SPLINE
SPL {X  -141.948, Y  +760.885, Z    +0.000, E1   -42.258, E3 +401984.281}
SPL {X  -160.264, Y  +717.397, Z    +0.000, E1   -24.835, E3 +402025.465}
SPL {X  -164.762, Y  +692.628, Z    +0.000, E1   -12.660, E3 +402028.718}
SPL {X  -165.581, Y  +680.274, Z    +0.000, E1    -5.699, E3 +402024.203}
SPL {X  -165.650, Y  +672.825, Z    +0.000, E1    -0.909, E3 +402022.391}
SPL {X  -165.650, Y  +667.803, Z    +0.000, E1    +2.989, E3 +402021.851}
SPL {X  -165.650, Y  +662.773, Z    +0.000, E1    +7.549, E3 +402021.773}
SPL {X  -165.650, Y  +656.581, Z    +0.000, E1   +13.870, E3 +402019.823}
SPL {X  -165.650, Y  +648.120, Z    +0.000, E1   +22.794, E3 +402019.054}
SPL {X  -165.650, Y  +632.103, Z    +0.000, E1   +42.949, E3 +402006.012}
SPL {X  -165.650, Y  +608.448, Z    +0.000, E1   +47.265, E3 +402032.452}
SPL {X  -165.650, Y  +595.526, Z    +0.000, E1   +48.856, E3 +402046.310}
SPL {X  -165.650, Y  +568.828, Z    +0.000, E1   +48.639, E3 +402088.863}
ENDSPLINE

SPLINE
SPL {X  -165.650, Y  +586.972, Z    +0.000, E1   +40.422, E3 +402099.562}
ENDSPLINE

SPLINE
SPL {X  -165.650, Y  +585.370, Z    +0.000, E1   +38.910, E3 +402112.822}
SPL {X  -165.650, Y  +580.805, Z    +0.000, E1   +38.877, E3 +402124.444}
SPL {X  -165.650, Y  +575.679, Z    +0.000, E1   +38.947, E3 +402137.166}
SPL {X  -165.650, Y  +569.616, Z    +0.000, E1   +38.966, E3 +402152.325}
SPL {X  -165.650, Y  +564.364, Z    +0.000, E1   +38.909, E3 +402165.977}
SPL {X  -165.650, Y  +559.065, Z    +0.000, E1   +38.883, E3 +402179.555}
SPL {X  -165.650, Y  +552.770, Z    +0.000, E1   +38.963, E3 +402195.116}
SPL {X  -165.650, Y  +546.277, Z    +0.000, E1   +38.910, E3 +402211.858}
SPL {X  -165.650, Y  +540.151, Z    +0.000, E1   +38.996, E3 +402226.787}
SPL {X  -165.650, Y  +534.008, Z    +0.000, E1   +38.962, E3 +402242.629}
SPL {X  -165.650, Y  +528.320, Z    +0.000, E1   +38.809, E3 +402257.866}
SPL {X  -165.650, Y  +524.195, Z    +0.000, E1   +38.844, E3 +402268.042}
SPL {X  -165.650, Y  +520.666, Z    +0.000, E1   +39.043, E3 +402275.767}
ENDSPLINE

SPLINE
SPL {X  -165.650, Y  +539.854, Z    +0.000, E1   +28.090, E3 +402288.602}
ENDSPLINE

SPLINE
SPL {X  -165.650, Y  +534.443, Z    +0.000, E1   +28.969, E3 +402302.654}
SPL {X  -165.650, Y  +530.452, Z    +0.000, E1   +29.664, E3 +402312.387}
SPL {X  -165.650, Y  +525.298, Z    +0.000, E1   +30.602, E3 +402324.197}
SPL {X  -165.650, Y  +518.290, Z    +0.000, E1   +31.783, E3 +402340.090}
SPL {X  -165.650, Y  +512.706, Z    +0.000, E1   +32.573, E3 +402352.924}
SPL {X  -165.650, Y  +507.785, Z    +0.000, E1   +33.438, E3 +402362.861}
SPL {X  -165.650, Y  +501.257, Z    +0.000, E1   +34.478, E3 +402376.101}
SPL {X  -165.650, Y  +493.800, Z    +0.000, E1   +35.486, E3 +402391.589}
SPL {X  -165.650, Y  +485.583, Z    +0.000, E1   +36.670, E3 +402407.312}
SPL {X  -165.650, Y  +477.375, Z    +0.000, E1   +37.747, E3 +402422.831}
SPL {X  -165.650, Y  +469.901, Z    +0.000, E1   +38.767, E3 +402435.963}
SPL {X  -165.650, Y  +461.805, Z    +0.000, E1   +39.619, E3 +402451.306}
SPL {X  -165.650, Y  +455.681, Z    +0.000, E1   +39.641, E3 +402466.095}
SPL {X  -165.650, Y  +451.332, Z    +0.000, E1   +39.738, E3 +402476.227}
SPL {X  -165.650, Y  +448.050, Z    +0.000, E1   +39.392, E3 +402486.393}
SPL {X  -165.650, Y  +442.946, Z    +0.000, E1   +39.866, E3 +402496.168}
SPL {X  -165.650, Y  +439.091, Z    +0.000, E1   +39.674, E3 +402506.786}
SPL {X  -165.650, Y  +434.131, Z    +0.000, E1   +39.643, E3 +402519.298}
SPL {X  -165.650, Y  +428.810, Z    +0.000, E1   +39.691, E3 +402532.060}
SPL {X  -165.650, Y  +424.197, Z    +0.000, E1   +39.695, E3 +402543.419}
SPL {X  -165.650, Y  +420.220, Z    +0.000, E1   +39.526, E3 +402554.214}
SPL {X  -165.650, Y  +414.177, Z    +0.000, E1   +39.693, E3 +402568.341}
SPL {X  -165.650, Y  +407.394, Z    +0.000, E1   +39.797, E3 +402584.296}
SPL {X  -165.650, Y  +402.798, Z    +0.000, E1   +39.651, E3 +402596.417}
SPL {X  -165.650, Y  +398.253, Z    +0.000, E1   +39.688, E3 +402607.421}
SPL {X  -165.650, Y  +393.720, Z    +0.000, E1   +39.686, E3 +402618.595}
SPL {X  -165.650, Y  +389.210, Z    +0.000, E1   +39.696, E3 +402629.645}
SPL {X  -165.650, Y  +384.878, Z    +0.000, E1   +39.631, E3 +402640.721}
SPL {X  -165.650, Y  +380.529, Z    +0.000, E1   +39.528, E3 +402652.108}
SPL {X  -165.618, Y  +375.240, Z    +0.000, E1   +39.617, E3 +402664.702}
SPL {X  -165.428, Y  +369.922, Z    +0.000, E1   +39.705, E3 +402677.243}
SPL {X  -165.216, Y  +366.519, Z    +0.000, E1   +39.498, E3 +402686.810}
SPL {X  -164.790, Y  +361.646, Z    +0.000, E1   +39.684, E3 +402697.805}
SPL {X  -164.317, Y  +357.530, Z    +0.000, E1   +39.402, E3 +402709.518}
SPL {X  -163.775, Y  +353.645, Z    +0.000, E1   +39.313, E3 +402719.689}
SPL {X  -162.932, Y  +348.615, Z    +0.000, E1   +39.259, E3 +402732.453}
SPL {X  -162.143, Y  +344.596, Z    +0.000, E1   +39.019, E3 +402743.670}
SPL {X  -161.093, Y  +339.912, Z    +0.000, E1   +38.966, E3 +402755.620}
SPL {X  -159.926, Y  +335.332, Z    +0.000, E1   +38.809, E3 +402767.674}
SPL {X  -154.584, Y  +318.971, Z    +0.000, E1   +44.936, E3 +402770.305}
SPL {X  -151.650, Y  +311.851, Z    +0.000, E1   +46.071, E3 +402777.840}
SPL {X  -148.632, Y  +305.368, Z    +0.000, E1   +40.700, E3 +402834.007}
SPL {X  -145.004, Y  +298.414, Z    +0.000, E1   +40.971, E3 +402858.743}
ENDSPLINE

SPLINE
SPL {X  -149.687, Y  +307.551, Z    +0.000, E1   +36.303, E3 +402894.175}
SPL {X  -158.807, Y  +331.381, Z    +0.000, E1   +26.928, E3 +402917.827}
SPL {X  -164.505, Y  +359.058, Z    +0.000, E1   +13.887, E3 +402906.589}
SPL {X  -165.494, Y  +371.321, Z    +0.000, E1    +7.176, E3 +402905.150}
SPL {X  -165.650, Y  +379.419, Z    +0.000, E1    +2.065, E3 +402902.831}
SPL {X  -165.650, Y  +383.176, Z    +0.000, E1    -0.610, E3 +402903.826}
SPL {X  -165.650, Y  +387.435, Z    +0.000, E1    -4.104, E3 +402902.186}
SPL {X  -165.650, Y  +393.422, Z    +0.000, E1    -9.605, E3 +402902.744}
SPL {X  -165.650, Y  +400.450, Z    +0.000, E1   -18.287, E3 +402894.558}
SPL {X  -165.650, Y  +409.248, Z    +0.000, E1   -26.478, E3 +402898.181}
SPL {X  -165.650, Y  +418.660, Z    +0.000, E1   -36.186, E3 +402895.657}
SPL {X  -165.650, Y  +444.260, Z    +0.000, E1   -47.328, E3 +402911.405}
SPL {X  -165.650, Y  +458.981, Z    +0.000, E1   -49.189, E3 +402926.948}
SPL {X  -165.650, Y  +493.049, Z    +0.000, E1   -51.657, E3 +402965.981}
ENDSPLINE

SPLINE
SPL {X  -165.650, Y  +468.984, Z    +0.000, E1   -41.461, E3 +402978.841}
SPL {X  -165.650, Y  +467.052, Z    +0.000, E1   -38.928, E3 +402989.456}
ENDSPLINE

SPLINE
SPL {X  -165.650, Y  +471.956, Z    +0.000, E1   -39.047, E3 +403001.107}
SPL {X  -165.650, Y  +476.270, Z    +0.000, E1   -39.142, E3 +403011.364}
SPL {X  -165.650, Y  +480.876, Z    +0.000, E1   -39.050, E3 +403023.646}
SPL {X  -165.650, Y  +487.054, Z    +0.000, E1   -39.118, E3 +403038.785}
SPL {X  -165.650, Y  +493.422, Z    +0.000, E1   -39.176, E3 +403054.507}
SPL {X  -165.650, Y  +499.941, Z    +0.000, E1   -39.068, E3 +403071.558}
SPL {X  -165.650, Y  +505.989, Z    +0.000, E1   -39.067, E3 +403086.738}
SPL {X  -165.650, Y  +512.188, Z    +0.000, E1   -39.077, E3 +403102.380}
SPL {X  -165.650, Y  +516.634, Z    +0.000, E1   -39.035, E3 +403113.626}
SPL {X  -165.650, Y  +521.541, Z    +0.000, E1   -39.052, E3 +403126.173}
SPL {X  -165.650, Y  +527.474, Z    +0.000, E1   -39.169, E3 +403140.191}
SPL {X  -165.650, Y  +532.836, Z    +0.000, E1   -39.150, E3 +403153.973}
SPL {X  -165.650, Y  +537.667, Z    +0.000, E1   -38.986, E3 +403166.918}
SPL {X  -165.650, Y  +541.183, Z    +0.000, E1   -39.101, E3 +403175.105}
SPL {X  -165.650, Y  +546.018, Z    +0.000, E1   -39.065, E3 +403187.616}
SPL {X  -165.650, Y  +551.666, Z    +0.000, E1   -39.102, E3 +403201.565}
SPL {X  -165.650, Y  +557.612, Z    +0.000, E1   -39.166, E3 +403216.211}
SPL {X  -165.650, Y  +562.850, Z    +0.000, E1   -38.959, E3 +403230.570}
SPL {X  -165.650, Y  +568.257, Z    +0.000, E1   -39.077, E3 +403243.525}
SPL {X  -165.650, Y  +573.200, Z    +0.000, E1   -39.061, E3 +403256.060}
SPL {X  -165.650, Y  +578.240, Z    +0.000, E1   -39.117, E3 +403268.401}
SPL {X  -165.650, Y  +582.804, Z    +0.000, E1   -39.080, E3 +403280.108}
SPL {X  -165.650, Y  +587.640, Z    +0.000, E1   -39.069, E3 +403292.365}
SPL {X  -165.650, Y  +593.610, Z    +0.000, E1   -39.204, E3 +403306.639}
SPL {X  -165.650, Y  +599.021, Z    +0.000, E1   -38.950, E3 +403321.788}
SPL {X  -165.650, Y  +604.635, Z    +0.000, E1   -39.163, E3 +403334.565}
SPL {X  -165.650, Y  +608.365, Z    +0.000, E1   -39.063, E3 +403344.555}
SPL {X  -165.650, Y  +612.142, Z    +0.000, E1   -39.023, E3 +403354.285}
SPL {X  -165.650, Y  +616.635, Z    +0.000, E1   -39.260, E3 +403364.172}
SPL {X  -165.650, Y  +620.299, Z    +0.000, E1   -38.904, E3 +403375.559}
SPL {X  -165.650, Y  +625.662, Z    +0.000, E1   -39.189, E3 +403387.370}
SPL {X  -165.650, Y  +629.982, Z    +0.000, E1   -39.063, E3 +403398.971}
SPL {X  -165.650, Y  +634.317, Z    +0.000, E1   -39.239, E3 +403408.762}
SPL {X  -165.650, Y  +639.215, Z    +0.000, E1   -39.074, E3 +403422.287}
SPL {X  -165.650, Y  +643.707, Z    +0.000, E1   -38.911, E3 +403434.387}
SPL {X  -165.650, Y  +648.294, Z    +0.000, E1   -39.142, E3 +403444.643}
SPL {X  -165.650, Y  +652.477, Z    +0.000, E1   -39.068, E3 +403455.545}
SPL {X  -165.650, Y  +656.920, Z    +0.000, E1   -39.120, E3 +403466.500}
SPL {X  -165.650, Y  +662.945, Z    +0.000, E1   -39.141, E3 +403481.605}
SPL {X  -165.650, Y  +668.296, Z    +0.000, E1   -39.077, E3 +403495.330}
SPL {X  -165.650, Y  +674.193, Z    +0.000, E1   -39.034, E3 +403510.672}
SPL {X  -165.521, Y  +682.029, Z    +0.000, E1   -39.160, E3 +403529.640}
SPL {X  -165.241, Y  +687.126, Z    +0.000, E1   -39.221, E3 +403541.802}
SPL {X  -164.948, Y  +690.736, Z    +0.000, E1   -38.951, E3 +403552.654}
SPL {X  -164.363, Y  +696.109, Z    +0.000, E1   -38.853, E3 +403566.745}
SPL {X  -163.795, Y  +700.218, Z    +0.000, E1   -38.698, E3 +403577.952}
SPL {X  -162.937, Y  +705.358, Z    +0.000, E1   -38.703, E3 +403591.020}
SPL {X  -161.983, Y  +710.160, Z    +0.000, E1   -38.439, E3 +403604.514}
SPL {X  -161.163, Y  +713.794, Z    +0.000, E1   -38.390, E3 +403613.884}
SPL {X  -160.616, Y  +716.027, Z    +0.000, E1   -37.944, E3 +403622.086}
SPL {X  -158.364, Y  +724.087, Z    +0.000, E1   -39.961, E3 +403630.382}
SPL {X  -138.706, Y  +766.057, Z    +0.000, E1   -46.957, E3 +403681.373}
ENDSPLINE

SPLINE
SPL {X  -141.948, Y  +760.885, Z    +0.000, E1   -42.258, E3 +403721.123}
SPL {X  -152.484, Y  +740.219, Z    +0.000, E1   -33.928, E3 +403758.276}
SPL {X  -161.203, Y  +713.624, Z    +0.000, E1   -23.097, E3 +403762.692}
SPL {X  -164.762, Y  +692.628, Z    +0.000, E1   -12.660, E3 +403765.560}
SPL {X  -165.581, Y  +680.274, Z    +0.000, E1    -5.699, E3 +403761.045}
SPL {X  -165.650, Y  +672.825, Z    +0.000, E1    -0.909, E3 +403759.234}
SPL {X  -165.650, Y  +667.803, Z    +0.000, E1    +2.989, E3 +403758.694}
SPL {X  -165.650, Y  +662.773, Z    +0.000, E1    +7.549, E3 +403758.615}
SPL {X  -165.650, Y  +656.581, Z    +0.000, E1   +13.870, E3 +403756.665}
SPL {X  -165.650, Y  +648.120, Z    +0.000, E1   +22.794, E3 +403755.896}
SPL {X  -165.650, Y  +632.103, Z    +0.000, E1   +42.949, E3 +403742.854}
SPL {X  -165.650, Y  +608.448, Z    +0.000, E1   +47.265, E3 +403769.294}
SPL {X  -165.650, Y  +595.526, Z    +0.000, E1   +48.856, E3 +403783.152}
SPL {X  -165.650, Y  +568.828, Z    +0.000, E1   +48.639, E3 +403825.705}
ENDSPLINE

SPLINE
SPL {X  -165.650, Y  +586.972, Z    +0.000, E1   +40.422, E3 +403836.404}
ENDSPLINE

SPLINE
SPL {X  -165.650, Y  +585.370, Z    +0.000, E1   +38.910, E3 +403849.664}
SPL {X  -165.650, Y  +580.805, Z    +0.000, E1   +38.877, E3 +403861.286}
SPL {X  -165.650, Y  +575.679, Z    +0.000, E1   +38.947, E3 +403874.009}
SPL {X  -165.650, Y  +569.616, Z    +0.000, E1   +38.966, E3 +403889.167}
SPL {X  -165.650, Y  +564.364, Z    +0.000, E1   +38.909, E3 +403902.820}
SPL {X  -165.650, Y  +559.065, Z    +0.000, E1   +38.883, E3 +403916.397}
SPL {X  -165.650, Y  +554.358, Z    +0.000, E1   +38.887, E3 +403928.239}
SPL {X  -165.650, Y  +549.409, Z    +0.000, E1   +38.884, E3 +403940.920}
SPL {X  -165.650, Y  +544.480, Z    +0.000, E1   +38.998, E3 +403952.584}
SPL {X  -165.650, Y  +540.151, Z    +0.000, E1   +38.996, E3 +403963.630}
SPL {X  -165.650, Y  +534.008, Z    +0.000, E1   +38.962, E3 +403979.472}
SPL {X  -165.650, Y  +528.320, Z    +0.000, E1   +38.809, E3 +403994.708}
SPL {X  -165.650, Y  +524.195, Z    +0.000, E1   +38.844, E3 +404004.884}
SPL {X  -165.650, Y  +520.666, Z    +0.000, E1   +39.043, E3 +404012.610}
ENDSPLINE

SPLINE
SPL {X  -165.650, Y  +541.168, Z    +0.000, E1   +27.957, E3 +404021.167}
ENDSPLINE

SPLINE
SPL {X  -165.650, Y  +536.052, Z    +0.000, E1   +28.653, E3 +404035.802}
SPL {X  -165.650, Y  +530.452, Z    +0.000, E1   +29.664, E3 +404049.229}
SPL {X  -165.650, Y  +523.712, Z    +0.000, E1   +30.911, E3 +404064.511}
SPL {X  -165.650, Y  +516.975, Z    +0.000, E1   +31.942, E3 +404080.105}
SPL {X  -165.650, Y  +512.706, Z    +0.000, E1   +32.573, E3 +404089.766}
SPL {X  -165.650, Y  +507.785, Z    +0.000, E1   +33.438, E3 +404099.703}
SPL {X  -165.650, Y  +501.257, Z    +0.000, E1   +34.478, E3 +404112.943}
SPL {X  -165.650, Y  +495.236, Z    +0.000, E1   +35.288, E3 +404125.449}
SPL {X  -165.650, Y  +488.684, Z    +0.000, E1   +36.217, E3 +404138.345}
SPL {X  -165.650, Y  +481.130, Z    +0.000, E1   +37.251, E3 +404152.654}
SPL {X  -165.650, Y  +475.455, Z    +0.000, E1   +37.964, E3 +404163.311}
SPL {X  -165.650, Y  +469.901, Z    +0.000, E1   +38.767, E3 +404172.805}
SPL {X  -165.650, Y  +465.276, Z    +0.000, E1   +39.067, E3 +404182.682}
SPL {X  -165.650, Y  +459.623, Z    +0.000, E1   +39.919, E3 +404191.617}
SPL {X  -165.650, Y  +455.681, Z    +0.000, E1   +39.641, E3 +404202.937}
SPL {X  -165.650, Y  +451.332, Z    +0.000, E1   +39.738, E3 +404213.069}
SPL {X  -165.650, Y  +448.050, Z    +0.000, E1   +39.392, E3 +404223.235}
SPL {X  -165.650, Y  +442.946, Z    +0.000, E1   +39.866, E3 +404233.010}
SPL {X  -165.650, Y  +439.091, Z    +0.000, E1   +39.674, E3 +404243.628}
SPL {X  -165.650, Y  +435.404, Z    +0.000, E1   +39.549, E3 +404253.465}
SPL {X  -165.650, Y  +429.757, Z    +0.000, E1   +39.737, E3 +404266.414}
SPL {X  -165.650, Y  +424.197, Z    +0.000, E1   +39.695, E3 +404280.261}
SPL {X  -165.650, Y  +420.220, Z    +0.000, E1   +39.526, E3 +404291.056}
SPL {X  -165.650, Y  +415.675, Z    +0.000, E1   +39.706, E3 +404301.218}
SPL {X  -165.650, Y  +410.648, Z    +0.000, E1   +39.653, E3 +404314.019}
SPL {X  -165.650, Y  +403.851, Z    +0.000, E1   +39.774, E3 +404330.104}
SPL {X  -165.650, Y  +398.253, Z    +0.000, E1   +39.688, E3 +404344.263}
SPL {X  -165.650, Y  +393.720, Z    +0.000, E1   +39.686, E3 +404355.437}
SPL {X  -165.650, Y  +389.210, Z    +0.000, E1   +39.696, E3 +404366.487}
SPL {X  -165.650, Y  +384.878, Z    +0.000, E1   +39.631, E3 +404377.564}
SPL {X  -165.650, Y  +380.529, Z    +0.000, E1   +39.528, E3 +404388.950}
SPL {X  -165.618, Y  +375.240, Z    +0.000, E1   +39.617, E3 +404401.544}
SPL {X  -165.428, Y  +369.922, Z    +0.000, E1   +39.705, E3 +404414.086}
SPL {X  -165.055, Y  +364.469, Z    +0.000, E1   +39.623, E3 +404428.127}
SPL {X  -164.424, Y  +358.387, Z    +0.000, E1   +39.525, E3 +404443.651}
SPL {X  -163.775, Y  +353.645, Z    +0.000, E1   +39.313, E3 +404456.531}
SPL {X  -162.932, Y  +348.615, Z    +0.000, E1   +39.259, E3 +404469.295}
SPL {X  -161.858, Y  +343.258, Z    +0.000, E1   +39.040, E3 +404483.834}
SPL {X  -160.812, Y  +338.758, Z    +0.000, E1   +38.898, E3 +404495.559}
SPL {X  -159.926, Y  +335.332, Z    +0.000, E1   +38.809, E3 +404504.516}
SPL {X  -153.020, Y  +315.059, Z    +0.000, E1   +45.580, E3 +404511.248}
SPL {X  -148.632, Y  +305.368, Z    +0.000, E1   +40.700, E3 +404570.849}
SPL {X  -145.004, Y  +298.414, Z    +0.000, E1   +40.971, E3 +404595.585}
ENDSPLINE

SPLINE
SPL {X  -149.687, Y  +307.551, Z    +0.000, E1   +36.303, E3 +404631.017}
SPL {X  -158.807, Y  +331.381, Z    +0.000, E1   +26.928, E3 +404654.670}
SPL {X  -164.505, Y  +359.058, Z    +0.000, E1   +13.887, E3 +404643.431}
SPL {X  -165.334, Y  +368.271, Z    +0.000, E1    +8.886, E3 +404641.270}
SPL {X  -165.596, Y  +374.277, Z    +0.000, E1    +5.306, E3 +404642.652}
SPL {X  -165.650, Y  +379.419, Z    +0.000, E1    +2.065, E3 +404639.673}
SPL {X  -165.650, Y  +383.176, Z    +0.000, E1    -0.610, E3 +404640.668}
SPL {X  -165.650, Y  +387.435, Z    +0.000, E1    -4.104, E3 +404639.029}
SPL {X  -165.650, Y  +393.422, Z    +0.000, E1    -9.605, E3 +404639.586}
SPL {X  -165.650, Y  +400.450, Z    +0.000, E1   -18.287, E3 +404631.400}
SPL {X  -165.650, Y  +409.248, Z    +0.000, E1   -26.478, E3 +404635.023}
SPL {X  -165.650, Y  +418.660, Z    +0.000, E1   -36.186, E3 +404632.499}
SPL {X  -165.650, Y  +444.260, Z    +0.000, E1   -47.328, E3 +404648.247}
SPL {X  -165.650, Y  +458.981, Z    +0.000, E1   -49.189, E3 +404663.791}
SPL {X  -165.650, Y  +493.049, Z    +0.000, E1   -51.657, E3 +404702.823}
ENDSPLINE

SPLINE
SPL {X  -165.650, Y  +468.984, Z    +0.000, E1   -41.461, E3 +404715.684}
SPL {X  -165.650, Y  +467.052, Z    +0.000, E1   -38.928, E3 +404726.298}
ENDSPLINE

SPLINE
SPL {X  -165.650, Y  +471.956, Z    +0.000, E1   -39.047, E3 +404737.949}
SPL {X  -165.650, Y  +476.270, Z    +0.000, E1   -39.142, E3 +404748.206}
SPL {X  -165.650, Y  +479.585, Z    +0.000, E1   -39.047, E3 +404757.117}
SPL {X  -165.650, Y  +484.115, Z    +0.000, E1   -39.050, E3 +404768.595}
SPL {X  -165.650, Y  +490.374, Z    +0.000, E1   -39.169, E3 +404783.715}
SPL {X  -165.650, Y  +495.141, Z    +0.000, E1   -39.109, E3 +404795.871}
SPL {X  -165.650, Y  +497.824, Z    +0.000, E1   -38.944, E3 +404803.630}
SPL {X  -165.650, Y  +502.351, Z    +0.000, E1   -39.056, E3 +404814.513}
SPL {X  -165.650, Y  +508.180, Z    +0.000, E1   -39.157, E3 +404828.579}
SPL {X  -165.650, Y  +513.074, Z    +0.000, E1   -38.997, E3 +404841.796}
SPL {X  -165.650, Y  +518.439, Z    +0.000, E1   -39.071, E3 +404854.947}
SPL {X  -165.650, Y  +523.032, Z    +0.000, E1   -38.966, E3 +404867.083}
SPL {X  -165.650, Y  +528.401, Z    +0.000, E1   -39.135, E3 +404879.683}
SPL {X  -165.650, Y  +533.857, Z    +0.000, E1   -39.163, E3 +404893.189}
SPL {X  -165.650, Y  +539.651, Z    +0.000, E1   -39.087, E3 +404908.333}
SPL {X  -165.650, Y  +544.603, Z    +0.000, E1   -39.103, E3 +404920.509}
SPL {X  -165.650, Y  +547.280, Z    +0.000, E1   -38.965, E3 +404928.089}
SPL {X  -165.650, Y  +551.666, Z    +0.000, E1   -39.102, E3 +404938.407}
SPL {X  -165.650, Y  +555.880, Z    +0.000, E1   -39.094, E3 +404948.978}
SPL {X  -165.650, Y  +559.255, Z    +0.000, E1   -39.167, E3 +404957.014}
SPL {X  -165.650, Y  +562.850, Z    +0.000, E1   -38.959, E3 +404967.412}
SPL {X  -165.650, Y  +568.257, Z    +0.000, E1   -39.077, E3 +404980.367}
SPL {X  -165.650, Y  +573.200, Z    +0.000, E1   -39.061, E3 +404992.902}
SPL {X  -165.650, Y  +578.240, Z    +0.000, E1   -39.117, E3 +405005.243}
SPL {X  -165.650, Y  +582.804, Z    +0.000, E1   -39.080, E3 +405016.950}
SPL {X  -165.650, Y  +587.640, Z    +0.000, E1   -39.069, E3 +405029.207}
SPL {X  -165.650, Y  +592.685, Z    +0.000, E1   -39.263, E3 +405040.671}
SPL {X  -165.650, Y  +596.539, Z    +0.000, E1   -39.049, E3 +405051.661}
SPL {X  -165.650, Y  +599.973, Z    +0.000, E1   -38.814, E3 +405061.714}
SPL {X  -165.650, Y  +604.635, Z    +0.000, E1   -39.163, E3 +405071.407}
SPL {X  -165.650, Y  +608.365, Z    +0.000, E1   -39.063, E3 +405081.397}
SPL {X  -165.650, Y  +612.142, Z    +0.000, E1   -39.023, E3 +405091.127}
SPL {X  -165.650, Y  +616.635, Z    +0.000, E1   -39.260, E3 +405101.014}
SPL {X  -165.650, Y  +620.299, Z    +0.000, E1   -38.904, E3 +405112.401}
SPL {X  -165.650, Y  +625.662, Z    +0.000, E1   -39.189, E3 +405124.212}
SPL {X  -165.650, Y  +629.982, Z    +0.000, E1   -39.063, E3 +405135.813}
SPL {X  -165.650, Y  +635.019, Z    +0.000, E1   -39.106, E3 +405148.295}
SPL {X  -165.650, Y  +640.403, Z    +0.000, E1   -39.127, E3 +405161.691}
SPL {X  -165.650, Y  +643.707, Z    +0.000, E1   -38.911, E3 +405171.229}
SPL {X  -165.650, Y  +648.294, Z    +0.000, E1   -39.142, E3 +405181.485}
SPL {X  -165.650, Y  +652.477, Z    +0.000, E1   -39.068, E3 +405192.387}
SPL {X  -165.650, Y  +656.920, Z    +0.000, E1   -39.120, E3 +405203.342}
SPL {X  -165.650, Y  +662.945, Z    +0.000, E1   -39.141, E3 +405218.448}
SPL {X  -165.650, Y  +668.296, Z    +0.000, E1   -39.077, E3 +405232.172}
SPL {X  -165.650, Y  +674.193, Z    +0.000, E1   -39.034, E3 +405247.514}
SPL {X  -165.521, Y  +682.029, Z    +0.000, E1   -39.160, E3 +405266.483}
SPL {X  -165.241, Y  +687.126, Z    +0.000, E1   -39.221, E3 +405278.644}
SPL {X  -165.072, Y  +689.330, Z    +0.000, E1   -38.812, E3 +405286.692}
SPL {X  -164.582, Y  +694.282, Z    +0.000, E1   -38.975, E3 +405298.301}
SPL {X  -163.926, Y  +699.336, Z    +0.000, E1   -38.767, E3 +405312.279}
SPL {X  -163.214, Y  +703.806, Z    +0.000, E1   -38.755, E3 +405323.464}
SPL {X  -162.700, Y  +706.623, Z    +0.000, E1   -38.580, E3 +405331.576}
SPL {X  -161.983, Y  +710.160, Z    +0.000, E1   -38.439, E3 +405341.356}
SPL {X  -161.163, Y  +713.794, Z    +0.000, E1   -38.390, E3 +405350.726}
SPL {X  -160.158, Y  +717.801, Z    +0.000, E1   -38.225, E3 +405361.856}
SPL {X  -155.870, Y  +731.575, Z    +0.000, E1   -42.661, E3 +405369.319}
SPL {X  -137.799, Y  +767.431, Z    +0.000, E1   -46.550, E3 +405425.829}
ENDSPLINE

SPLINE
SPL {X  -141.948, Y  +760.885, Z    +0.000, E1   -42.258, E3 +405457.965}
SPL {X  -152.484, Y  +740.219, Z    +0.000, E1   -33.928, E3 +405495.119}
SPL {X  -161.203, Y  +713.624, Z    +0.000, E1   -23.097, E3 +405499.534}
SPL {X  -164.762, Y  +692.628, Z    +0.000, E1   -12.660, E3 +405502.402}
SPL {X  -165.481, Y  +682.990, Z    +0.000, E1    -7.255, E3 +405499.247}
SPL {X  -165.649, Y  +676.021, Z    +0.000, E1    -3.061, E3 +405496.614}
SPL {X  -165.650, Y  +670.589, Z    +0.000, E1    +0.778, E3 +405495.851}
SPL {X  -165.650, Y  +666.842, Z    +0.000, E1    +3.871, E3 +405495.312}
SPL {X  -165.650, Y  +662.773, Z    +0.000, E1    +7.549, E3 +405495.457}
SPL {X  -165.650, Y  +656.581, Z    +0.000, E1   +13.870, E3 +405493.507}
SPL {X  -165.650, Y  +648.120, Z    +0.000, E1   +22.794, E3 +405492.738}
SPL {X  -165.650, Y  +632.103, Z    +0.000, E1   +42.949, E3 +405479.696}
SPL {X  -165.650, Y  +608.448, Z    +0.000, E1   +47.265, E3 +405506.136}
SPL {X  -165.650, Y  +595.526, Z    +0.000, E1   +48.856, E3 +405519.994}
SPL {X  -165.650, Y  +568.828, Z    +0.000, E1   +48.639, E3 +405562.547}
ENDSPLINE

SPLINE
SPL {X  -165.650, Y  +586.972, Z    +0.000, E1   +40.422, E3 +405573.246}
ENDSPLINE

SPLINE
SPL {X  -165.650, Y  +585.370, Z    +0.000, E1   +38.910, E3 +405586.506}
SPL {X  -165.650, Y  +580.805, Z    +0.000, E1   +38.877, E3 +405598.128}
SPL {X  -165.650, Y  +575.679, Z    +0.000, E1   +38.947, E3 +405610.851}
SPL {X  -165.650, Y  +569.616, Z    +0.000, E1   +38.966, E3 +405626.009}
SPL {X  -165.650, Y  +564.364, Z    +0.000, E1   +38.909, E3 +405639.662}
SPL {X  -165.650, Y  +559.065, Z    +0.000, E1   +38.883, E3 +405653.240}
SPL {X  -165.650, Y  +552.770, Z    +0.000, E1   +38.963, E3 +405668.800}
SPL {X  -165.650, Y  +546.277, Z    +0.000, E1   +38.910, E3 +405685.542}
SPL {X  -165.650, Y  +541.194, Z    +0.000, E1   +39.037, E3 +405697.475}
SPL {X  -165.650, Y  +537.647, Z    +0.000, E1   +38.838, E3 +405707.720}
SPL {X  -165.650, Y  +532.636, Z    +0.000, E1   +39.009, E3 +405719.366}
SPL {X  -165.650, Y  +528.320, Z    +0.000, E1   +38.809, E3 +405731.550}
SPL {X  -165.650, Y  +522.377, Z    +0.000, E1   +38.974, E3 +405745.670}
ENDSPLINE

SPLINE
SPL {X  -165.650, Y  +541.168, Z    +0.000, E1   +27.957, E3 +405758.010}
ENDSPLINE

SPLINE
SPL {X  -165.650, Y  +536.052, Z    +0.000, E1   +28.653, E3 +405772.644}
SPL {X  -165.650, Y  +530.452, Z    +0.000, E1   +29.664, E3 +405786.071}
SPL {X  -165.650, Y  +523.712, Z    +0.000, E1   +30.911, E3 +405801.353}
SPL {X  -165.650, Y  +516.975, Z    +0.000, E1   +31.942, E3 +405816.947}
SPL {X  -165.650, Y  +512.706, Z    +0.000, E1   +32.573, E3 +405826.608}
SPL {X  -165.650, Y  +507.785, Z    +0.000, E1   +33.438, E3 +405836.546}
SPL {X  -165.650, Y  +502.877, Z    +0.000, E1   +34.230, E3 +405846.434}
SPL {X  -165.650, Y  +496.704, Z    +0.000, E1   +35.113, E3 +405859.227}
SPL {X  -165.650, Y  +488.684, Z    +0.000, E1   +36.217, E3 +405875.188}
SPL {X  -165.650, Y  +481.130, Z    +0.000, E1   +37.251, E3 +405889.497}
SPL {X  -165.650, Y  +475.455, Z    +0.000, E1   +37.964, E3 +405900.153}
SPL {X  -165.650, Y  +469.901, Z    +0.000, E1   +38.767, E3 +405909.647}
SPL {X  -165.650, Y  +461.805, Z    +0.000, E1   +39.619, E3 +405924.990}
SPL {X  -165.650, Y  +455.681, Z    +0.000, E1   +39.641, E3 +405939.779}
SPL {X  -165.650, Y  +451.332, Z    +0.000, E1   +39.738, E3 +405949.912}
SPL {X  -165.650, Y  +448.050, Z    +0.000, E1   +39.392, E3 +405960.077}
SPL {X  -165.650, Y  +442.946, Z    +0.000, E1   +39.866, E3 +405969.852}
SPL {X  -165.650, Y  +439.091, Z    +0.000, E1   +39.674, E3 +405980.470}
SPL {X  -165.650, Y  +434.131, Z    +0.000, E1   +39.643, E3 +405992.983}
SPL {X  -165.650, Y  +428.810, Z    +0.000, E1   +39.691, E3 +406005.745}
SPL {X  -165.650, Y  +424.197, Z    +0.000, E1   +39.695, E3 +406017.103}
SPL {X  -165.650, Y  +420.220, Z    +0.000, E1   +39.526, E3 +406027.898}
SPL {X  -165.650, Y  +414.177, Z    +0.000, E1   +39.693, E3 +406042.025}
SPL {X  -165.650, Y  +407.394, Z    +0.000, E1   +39.797, E3 +406057.980}
SPL {X  -165.650, Y  +402.798, Z    +0.000, E1   +39.651, E3 +406070.102}
SPL {X  -165.650, Y  +398.253, Z    +0.000, E1   +39.688, E3 +406081.105}
SPL {X  -165.650, Y  +393.720, Z    +0.000, E1   +39.686, E3 +406092.280}
SPL {X  -165.650, Y  +389.210, Z    +0.000, E1   +39.696, E3 +406103.329}
SPL {X  -165.650, Y  +384.878, Z    +0.000, E1   +39.631, E3 +406114.406}
SPL {X  -165.650, Y  +378.931, Z    +0.000, E1   +39.598, E3 +406129.502}
SPL {X  -165.490, Y  +371.216, Z    +0.000, E1   +39.708, E3 +406147.874}
SPL {X  -165.055, Y  +364.469, Z    +0.000, E1   +39.623, E3 +406164.969}
SPL {X  -164.424, Y  +358.387, Z    +0.000, E1   +39.525, E3 +406180.493}
SPL {X  -163.775, Y  +353.645, Z    +0.000, E1   +39.313, E3 +406193.373}
SPL {X  -162.932, Y  +348.615, Z    +0.000, E1   +39.259, E3 +406206.137}
SPL {X  -162.143, Y  +344.596, Z    +0.000, E1   +39.019, E3 +406217.354}
SPL {X  -161.093, Y  +339.912, Z    +0.000, E1   +38.966, E3 +406229.305}
SPL {X  -159.926, Y  +335.332, Z    +0.000, E1   +38.809, E3 +406241.358}
SPL {X  -153.020, Y  +315.059, Z    +0.000, E1   +45.580, E3 +406248.090}
SPL {X  -148.632, Y  +305.368, Z    +0.000, E1   +40.700, E3 +406307.692}
SPL {X  -145.004, Y  +298.414, Z    +0.000, E1   +40.971, E3 +406332.427}
ENDSPLINE

SPLINE
SPL {X  -149.687, Y  +307.551, Z    +0.000, E1   +36.303, E3 +406367.859}
SPL {X  -158.807, Y  +331.381, Z    +0.000, E1   +26.928, E3 +406391.512}
SPL {X  -164.505, Y  +359.058, Z    +0.000, E1   +13.887, E3 +406380.274}
SPL {X  -165.494, Y  +371.321, Z    +0.000, E1    +7.176, E3 +406378.834}
SPL {X  -165.650, Y  +379.419, Z    +0.000, E1    +2.065, E3 +406376.516}
SPL {X  -165.650, Y  +383.176, Z    +0.000, E1    -0.610, E3 +406377.511}
SPL {X  -165.650, Y  +388.696, Z    +0.000, E1    -5.134, E3 +406375.787}
SPL {X  -165.650, Y  +394.663, Z    +0.000, E1   -10.843, E3 +406376.943}
SPL {X  -165.650, Y  +400.450, Z    +0.000, E1   -18.287, E3 +406368.242}
SPL {X  -165.650, Y  +409.248, Z    +0.000, E1   -26.478, E3 +406371.865}
SPL {X  -165.650, Y  +418.660, Z    +0.000, E1   -36.186, E3 +406369.341}
SPL {X  -165.650, Y  +444.260, Z    +0.000, E1   -47.328, E3 +406385.089}
SPL {X  -165.650, Y  +458.981, Z    +0.000, E1   -49.189, E3 +406400.633}
SPL {X  -165.650, Y  +493.049, Z    +0.000, E1   -51.657, E3 +406439.665}
ENDSPLINE

SPLINE
SPL {X  -165.650, Y  +468.984, Z    +0.000, E1   -41.461, E3 +406452.526}
SPL {X  -165.650, Y  +467.052, Z    +0.000, E1   -38.928, E3 +406463.140}
ENDSPLINE

SPLINE
SPL {X  -165.650, Y  +471.956, Z    +0.000, E1   -39.047, E3 +406474.792}
SPL {X  -165.650, Y  +478.019, Z    +0.000, E1   -39.139, E3 +406489.676}
SPL {X  -165.650, Y  +484.115, Z    +0.000, E1   -39.050, E3 +406505.437}
SPL {X  -165.650, Y  +488.489, Z    +0.000, E1   -39.102, E3 +406516.046}
SPL {X  -165.650, Y  +491.785, Z    +0.000, E1   -39.157, E3 +406524.018}
SPL {X  -165.650, Y  +496.519, Z    +0.000, E1   -39.062, E3 +406536.632}
SPL {X  -165.650, Y  +501.480, Z    +0.000, E1   -39.099, E3 +406548.789}
SPL {X  -165.650, Y  +505.989, Z    +0.000, E1   -39.067, E3 +406560.422}
SPL {X  -165.650, Y  +512.188, Z    +0.000, E1   -39.077, E3 +406576.064}
SPL {X  -165.650, Y  +516.634, Z    +0.000, E1   -39.035, E3 +406587.310}
SPL {X  -165.650, Y  +521.541, Z    +0.000, E1   -39.052, E3 +406599.857}
SPL {X  -165.650, Y  +528.401, Z    +0.000, E1   -39.135, E3 +406616.526}
SPL {X  -165.650, Y  +533.857, Z    +0.000, E1   -39.163, E3 +406630.031}
SPL {X  -165.650, Y  +539.651, Z    +0.000, E1   -39.087, E3 +406645.175}
SPL {X  -165.650, Y  +544.603, Z    +0.000, E1   -39.103, E3 +406657.351}
SPL {X  -165.650, Y  +547.280, Z    +0.000, E1   -38.965, E3 +406664.931}
SPL {X  -165.650, Y  +551.666, Z    +0.000, E1   -39.102, E3 +406675.249}
SPL {X  -165.650, Y  +555.880, Z    +0.000, E1   -39.094, E3 +406685.820}
SPL {X  -165.650, Y  +559.255, Z    +0.000, E1   -39.167, E3 +406693.857}
SPL {X  -165.650, Y  +562.850, Z    +0.000, E1   -38.959, E3 +406704.254}
SPL {X  -165.650, Y  +568.257, Z    +0.000, E1   -39.077, E3 +406717.209}
SPL {X  -165.650, Y  +573.200, Z    +0.000, E1   -39.061, E3 +406729.744}
SPL {X  -165.650, Y  +578.240, Z    +0.000, E1   -39.117, E3 +406742.085}
SPL {X  -165.650, Y  +582.804, Z    +0.000, E1   -39.080, E3 +406753.792}
SPL {X  -165.650, Y  +587.640, Z    +0.000, E1   -39.069, E3 +406766.049}
SPL {X  -165.650, Y  +592.685, Z    +0.000, E1   -39.263, E3 +406777.513}
SPL {X  -165.650, Y  +596.539, Z    +0.000, E1   -39.049, E3 +406788.503}
SPL {X  -165.650, Y  +599.973, Z    +0.000, E1   -38.814, E3 +406798.556}
SPL {X  -165.650, Y  +604.635, Z    +0.000, E1   -39.163, E3 +406808.249}
SPL {X  -165.650, Y  +608.365, Z    +0.000, E1   -39.063, E3 +406818.239}
SPL {X  -165.650, Y  +612.142, Z    +0.000, E1   -39.023, E3 +406827.969}
SPL {X  -165.650, Y  +616.635, Z    +0.000, E1   -39.260, E3 +406837.857}
SPL {X  -165.650, Y  +620.299, Z    +0.000, E1   -38.904, E3 +406849.243}
SPL {X  -165.650, Y  +625.662, Z    +0.000, E1   -39.189, E3 +406861.054}
SPL {X  -165.650, Y  +629.982, Z    +0.000, E1   -39.063, E3 +406872.655}
SPL {X  -165.650, Y  +635.019, Z    +0.000, E1   -39.106, E3 +406885.137}
SPL {X  -165.650, Y  +640.403, Z    +0.000, E1   -39.127, E3 +406898.533}
SPL {X  -165.650, Y  +645.443, Z    +0.000, E1   -39.032, E3 +406911.838}
SPL {X  -165.650, Y  +651.452, Z    +0.000, E1   -39.128, E3 +406926.408}
SPL {X  -165.650, Y  +656.920, Z    +0.000, E1   -39.120, E3 +406940.184}
SPL {X  -165.650, Y  +662.945, Z    +0.000, E1   -39.141, E3 +406955.290}
SPL {X  -165.650, Y  +668.296, Z    +0.000, E1   -39.077, E3 +406969.015}
SPL {X  -165.650, Y  +674.193, Z    +0.000, E1   -39.034, E3 +406984.356}
SPL {X  -165.521, Y  +682.029, Z    +0.000, E1   -39.160, E3 +407003.325}
SPL {X  -165.241, Y  +687.126, Z    +0.000, E1   -39.221, E3 +407015.486}
SPL {X  -165.072, Y  +689.330, Z    +0.000, E1   -38.812, E3 +407023.534}
SPL {X  -164.582, Y  +694.282, Z    +0.000, E1   -38.975, E3 +407035.143}
SPL {X  -163.926, Y  +699.336, Z    +0.000, E1   -38.767, E3 +407049.121}
SPL {X  -163.214, Y  +703.806, Z    +0.000, E1   -38.755, E3 +407060.306}
SPL {X  -162.700, Y  +706.623, Z    +0.000, E1   -38.580, E3 +407068.419}
SPL {X  -161.983, Y  +710.160, Z    +0.000, E1   -38.439, E3 +407078.198}
SPL {X  -161.163, Y  +713.794, Z    +0.000, E1   -38.390, E3 +407087.568}
SPL {X  -160.158, Y  +717.801, Z    +0.000, E1   -38.225, E3 +407098.698}
SPL {X  -155.870, Y  +731.575, Z    +0.000, E1   -42.661, E3 +407106.161}
SPL {X  -137.799, Y  +767.431, Z    +0.000, E1   -46.550, E3 +407162.671}
ENDSPLINE

SPLINE
SPL {X  -141.948, Y  +760.885, Z    +0.000, E1   -42.258, E3 +407194.807}
SPL {X  -160.264, Y  +717.397, Z    +0.000, E1   -24.835, E3 +407235.992}
SPL {X  -164.762, Y  +692.628, Z    +0.000, E1   -12.660, E3 +407239.245}
SPL {X  -165.481, Y  +682.990, Z    +0.000, E1    -7.255, E3 +407236.089}
SPL {X  -165.650, Y  +675.052, Z    +0.000, E1    -2.475, E3 +407232.306}
SPL {X  -165.650, Y  +670.254, Z    +0.000, E1    +1.045, E3 +407234.052}
SPL {X  -165.650, Y  +666.842, Z    +0.000, E1    +3.871, E3 +407232.154}
SPL {X  -165.650, Y  +662.773, Z    +0.000, E1    +7.549, E3 +407232.299}
SPL {X  -165.650, Y  +656.581, Z    +0.000, E1   +13.870, E3 +407230.349}
SPL {X  -165.650, Y  +648.120, Z    +0.000, E1   +22.794, E3 +407229.580}
SPL {X  -165.650, Y  +632.103, Z    +0.000, E1   +42.949, E3 +407216.538}
SPL {X  -165.650, Y  +608.448, Z    +0.000, E1   +47.265, E3 +407242.978}
SPL {X  -165.650, Y  +595.526, Z    +0.000, E1   +48.856, E3 +407256.836}
SPL {X  -165.650, Y  +568.828, Z    +0.000, E1   +48.639, E3 +407299.389}
ENDSPLINE

SPLINE
SPL {X  -165.650, Y  +586.972, Z    +0.000, E1   +40.422, E3 +407310.088}
ENDSPLINE

SPLINE
SPL {X  -165.650, Y  +585.370, Z    +0.000, E1   +38.910, E3 +407323.348}
SPL {X  -165.650, Y  +580.805, Z    +0.000, E1   +38.877, E3 +407334.970}
SPL {X  -165.650, Y  +575.679, Z    +0.000, E1   +38.947, E3 +407347.693}
SPL {X  -165.650, Y  +569.616, Z    +0.000, E1   +38.966, E3 +407362.851}
SPL {X  -165.650, Y  +564.364, Z    +0.000, E1   +38.909, E3 +407376.504}
SPL {X  -165.650, Y  +559.065, Z    +0.000, E1   +38.883, E3 +407390.082}
SPL {X  -165.650, Y  +552.770, Z    +0.000, E1   +38.963, E3 +407405.642}
SPL {X  -165.650, Y  +548.337, Z    +0.000, E1   +38.743, E3 +407418.022}
SPL {X  -165.650, Y  +542.772, Z    +0.000, E1   +39.054, E3 +407430.400}
SPL {X  -165.650, Y  +537.647, Z    +0.000, E1   +38.838, E3 +407444.563}
SPL {X  -165.650, Y  +532.636, Z    +0.000, E1   +39.009, E3 +407456.209}
SPL {X  -165.650, Y  +528.320, Z    +0.000, E1   +38.809, E3 +407468.392}
SPL {X  -165.650, Y  +522.377, Z    +0.000, E1   +38.974, E3 +407482.512}
ENDSPLINE

SPLINE
SPL {X  -165.650, Y  +541.168, Z    +0.000, E1   +27.957, E3 +407494.852}
ENDSPLINE

SPLINE
SPL {X  -165.650, Y  +536.052, Z    +0.000, E1   +28.653, E3 +407509.486}
SPL {X  -165.650, Y  +530.452, Z    +0.000, E1   +29.664, E3 +407522.913}
SPL {X  -165.650, Y  +525.298, Z    +0.000, E1   +30.602, E3 +407534.724}
SPL {X  -165.650, Y  +518.290, Z    +0.000, E1   +31.783, E3 +407550.616}
SPL {X  -165.650, Y  +512.706, Z    +0.000, E1   +32.573, E3 +407563.450}
SPL {X  -165.650, Y  +507.785, Z    +0.000, E1   +33.438, E3 +407573.388}
SPL {X  -165.650, Y  +501.257, Z    +0.000, E1   +34.478, E3 +407586.627}
SPL {X  -165.650, Y  +495.236, Z    +0.000, E1   +35.288, E3 +407599.133}
SPL {X  -165.650, Y  +488.684, Z    +0.000, E1   +36.217, E3 +407612.030}
SPL {X  -165.650, Y  +481.130, Z    +0.000, E1   +37.251, E3 +407626.339}
SPL {X  -165.650, Y  +475.455, Z    +0.000, E1   +37.964, E3 +407636.995}
SPL {X  -165.650, Y  +469.901, Z    +0.000, E1   +38.767, E3 +407646.489}
SPL {X  -165.650, Y  +461.805, Z    +0.000, E1   +39.619, E3 +407661.832}
SPL {X  -165.650, Y  +455.681, Z    +0.000, E1   +39.641, E3 +407676.621}
SPL {X  -165.650, Y  +451.332, Z    +0.000, E1   +39.738, E3 +407686.754}
SPL {X  -165.650, Y  +448.050, Z    +0.000, E1   +39.392, E3 +407696.920}
SPL {X  -165.650, Y  +442.946, Z    +0.000, E1   +39.866, E3 +407706.694}
SPL {X  -165.650, Y  +439.091, Z    +0.000, E1   +39.674, E3 +407717.312}
SPL {X  -165.650, Y  +434.131, Z    +0.000, E1   +39.643, E3 +407729.825}
SPL {X  -165.650, Y  +428.810, Z    +0.000, E1   +39.691, E3 +407742.587}
SPL {X  -165.650, Y  +424.197, Z    +0.000, E1   +39.695, E3 +407753.945}
SPL {X  -165.650, Y  +420.220, Z    +0.000, E1   +39.526, E3 +407764.741}
SPL {X  -165.650, Y  +414.177, Z    +0.000, E1   +39.693, E3 +407778.867}
SPL {X  -165.650, Y  +407.394, Z    +0.000, E1   +39.797, E3 +407794.822}
SPL {X  -165.650, Y  +402.798, Z    +0.000, E1   +39.651, E3 +407806.944}
SPL {X  -165.650, Y  +398.253, Z    +0.000, E1   +39.688, E3 +407817.947}
SPL {X  -165.650, Y  +393.720, Z    +0.000, E1   +39.686, E3 +407829.122}
SPL {X  -165.650, Y  +389.210, Z    +0.000, E1   +39.696, E3 +407840.171}
SPL {X  -165.650, Y  +384.878, Z    +0.000, E1   +39.631, E3 +407851.248}
SPL {X  -165.650, Y  +380.529, Z    +0.000, E1   +39.528, E3 +407862.634}
SPL {X  -165.618, Y  +375.240, Z    +0.000, E1   +39.617, E3 +407875.228}
SPL {X  -165.428, Y  +369.922, Z    +0.000, E1   +39.705, E3 +407887.770}
SPL {X  -165.216, Y  +366.519, Z    +0.000, E1   +39.498, E3 +407897.337}
SPL {X  -164.790, Y  +361.646, Z    +0.000, E1   +39.684, E3 +407908.331}
SPL {X  -164.317, Y  +357.530, Z    +0.000, E1   +39.402, E3 +407920.044}
SPL {X  -163.775, Y  +353.645, Z    +0.000, E1   +39.313, E3 +407930.215}
SPL {X  -163.109, Y  +349.595, Z    +0.000, E1   +39.290, E3 +407940.277}
SPL {X  -162.309, Y  +345.398, Z    +0.000, E1   +39.085, E3 +407951.941}
SPL {X  -161.467, Y  +341.510, Z    +0.000, E1   +38.980, E3 +407961.986}
SPL {X  -160.812, Y  +338.758, Z    +0.000, E1   +38.898, E3 +407969.243}
SPL {X  -159.926, Y  +335.332, Z    +0.000, E1   +38.809, E3 +407978.201}
SPL {X  -153.020, Y  +315.059, Z    +0.000, E1   +45.580, E3 +407984.932}
SPL {X  -148.632, Y  +305.368, Z    +0.000, E1   +40.700, E3 +408044.534}
SPL {X  -145.004, Y  +298.414, Z    +0.000, E1   +40.971, E3 +408069.269}
ENDSPLINE

SPLINE
SPL {X  -149.687, Y  +307.551, Z    +0.000, E1   +36.303, E3 +408104.701}
SPL {X  -158.807, Y  +331.381, Z    +0.000, E1   +26.928, E3 +408128.354}
SPL {X  -164.505, Y  +359.058, Z    +0.000, E1   +13.887, E3 +408117.116}
SPL {X  -165.494, Y  +371.321, Z    +0.000, E1    +7.176, E3 +408115.676}
SPL {X  -165.650, Y  +379.419, Z    +0.000, E1    +2.065, E3 +408113.358}
SPL {X  -165.650, Y  +383.176, Z    +0.000, E1    -0.610, E3 +408114.353}
SPL {X  -165.650, Y  +387.435, Z    +0.000, E1    -4.104, E3 +408112.713}
SPL {X  -165.650, Y  +393.422, Z    +0.000, E1    -9.605, E3 +408113.270}
SPL {X  -165.650, Y  +400.450, Z    +0.000, E1   -18.287, E3 +408105.084}
SPL {X  -165.650, Y  +409.248, Z    +0.000, E1   -26.478, E3 +408108.707}
SPL {X  -165.650, Y  +418.660, Z    +0.000, E1   -36.186, E3 +408106.183}
SPL {X  -165.650, Y  +444.260, Z    +0.000, E1   -47.328, E3 +408121.931}
SPL {X  -165.650, Y  +458.981, Z    +0.000, E1   -49.189, E3 +408137.475}
SPL {X  -165.650, Y  +493.049, Z    +0.000, E1   -51.657, E3 +408176.508}
ENDSPLINE

SPLINE
SPL {X  -165.650, Y  +468.984, Z    +0.000, E1   -41.461, E3 +408189.368}
SPL {X  -165.650, Y  +467.052, Z    +0.000, E1   -38.928, E3 +408199.983}
ENDSPLINE

SPLINE
SPL {X  -165.650, Y  +471.956, Z    +0.000, E1   -39.047, E3 +408211.634}
SPL {X  -165.650, Y  +476.270, Z    +0.000, E1   -39.142, E3 +408221.890}
SPL {X  -165.650, Y  +480.876, Z    +0.000, E1   -39.050, E3 +408234.172}
SPL {X  -165.650, Y  +487.054, Z    +0.000, E1   -39.118, E3 +408249.311}
SPL {X  -165.650, Y  +491.785, Z    +0.000, E1   -39.157, E3 +408260.860}
SPL {X  -165.650, Y  +496.519, Z    +0.000, E1   -39.062, E3 +408273.474}
SPL {X  -165.650, Y  +502.351, Z    +0.000, E1   -39.056, E3 +408288.197}
SPL {X  -165.650, Y  +508.180, Z    +0.000, E1   -39.157, E3 +408302.263}
SPL {X  -165.650, Y  +513.074, Z    +0.000, E1   -38.997, E3 +408315.481}
SPL {X  -165.650, Y  +518.439, Z    +0.000, E1   -39.071, E3 +408328.631}
SPL {X  -165.650, Y  +523.032, Z    +0.000, E1   -38.966, E3 +408340.767}
SPL {X  -165.650, Y  +528.401, Z    +0.000, E1   -39.135, E3 +408353.368}
SPL {X  -165.650, Y  +533.857, Z    +0.000, E1   -39.163, E3 +408366.873}
SPL {X  -165.650, Y  +539.651, Z    +0.000, E1   -39.087, E3 +408382.017}
SPL {X  -165.650, Y  +546.018, Z    +0.000, E1   -39.065, E3 +408398.142}
SPL {X  -165.650, Y  +551.666, Z    +0.000, E1   -39.102, E3 +408412.091}
SPL {X  -165.650, Y  +557.612, Z    +0.000, E1   -39.166, E3 +408426.738}
SPL {X  -165.650, Y  +562.850, Z    +0.000, E1   -38.959, E3 +408441.096}
SPL {X  -165.650, Y  +568.257, Z    +0.000, E1   -39.077, E3 +408454.051}
SPL {X  -165.650, Y  +573.200, Z    +0.000, E1   -39.061, E3 +408466.586}
SPL {X  -165.650, Y  +578.240, Z    +0.000, E1   -39.117, E3 +408478.927}
SPL {X  -165.650, Y  +582.804, Z    +0.000, E1   -39.080, E3 +408490.634}
SPL {X  -165.650, Y  +587.640, Z    +0.000, E1   -39.069, E3 +408502.891}
SPL {X  -165.650, Y  +593.610, Z    +0.000, E1   -39.204, E3 +408517.165}
SPL {X  -165.650, Y  +599.021, Z    +0.000, E1   -38.950, E3 +408532.314}
SPL {X  -165.650, Y  +604.635, Z    +0.000, E1   -39.163, E3 +408545.091}
SPL {X  -165.650, Y  +608.365, Z    +0.000, E1   -39.063, E3 +408555.081}
SPL {X  -165.650, Y  +613.618, Z    +0.000, E1   -39.137, E3 +408567.945}
SPL {X  -165.650, Y  +619.584, Z    +0.000, E1   -39.045, E3 +408583.582}
SPL {X  -165.650, Y  +625.662, Z    +0.000, E1   -39.189, E3 +408597.896}
SPL {X  -165.650, Y  +629.982, Z    +0.000, E1   -39.063, E3 +408609.498}
SPL {X  -165.650, Y  +635.019, Z    +0.000, E1   -39.106, E3 +408621.980}
SPL {X  -165.650, Y  +640.403, Z    +0.000, E1   -39.127, E3 +408635.375}
SPL {X  -165.650, Y  +645.443, Z    +0.000, E1   -39.032, E3 +408648.680}
SPL {X  -165.650, Y  +651.452, Z    +0.000, E1   -39.128, E3 +408663.250}
SPL {X  -165.650, Y  +656.920, Z    +0.000, E1   -39.120, E3 +408677.027}
SPL {X  -165.650, Y  +662.945, Z    +0.000, E1   -39.141, E3 +408692.132}
SPL {X  -165.650, Y  +668.296, Z    +0.000, E1   -39.077, E3 +408705.857}
SPL {X  -165.650, Y  +673.138, Z    +0.000, E1   -39.196, E3 +408717.313}
SPL {X  -165.640, Y  +677.281, Z    +0.000, E1   -38.803, E3 +408730.201}
SPL {X  -165.461, Y  +683.414, Z    +0.000, E1   -39.212, E3 +408743.185}
SPL {X  -165.139, Y  +688.497, Z    +0.000, E1   -39.013, E3 +408757.237}
SPL {X  -164.582, Y  +694.282, Z    +0.000, E1   -38.975, E3 +408771.985}
SPL {X  -163.926, Y  +699.336, Z    +0.000, E1   -38.767, E3 +408785.963}
SPL {X  -162.937, Y  +705.358, Z    +0.000, E1   -38.703, E3 +408801.547}
SPL {X  -161.983, Y  +710.160, Z    +0.000, E1   -38.439, E3 +408815.040}
SPL {X  -160.874, Y  +714.989, Z    +0.000, E1   -38.205, E3 +408828.702}
SPL {X  -158.364, Y  +724.087, Z    +0.000, E1   -39.961, E3 +408840.908}
SPL {X  -138.706, Y  +766.057, Z    +0.000, E1   -46.957, E3 +408891.899}
ENDSPLINE

SPLINE
SPL {X  -141.948, Y  +760.885, Z    +0.000, E1   -42.258, E3 +408931.649}
SPL {X  -160.264, Y  +717.397, Z    +0.000, E1   -24.835, E3 +408972.834}
SPL {X  -164.762, Y  +692.628, Z    +0.000, E1   -12.660, E3 +408976.087}
SPL {X  -165.581, Y  +680.274, Z    +0.000, E1    -5.699, E3 +408971.571}
SPL {X  -165.650, Y  +672.825, Z    +0.000, E1    -0.909, E3 +408969.760}
SPL {X  -165.650, Y  +667.803, Z    +0.000, E1    +2.989, E3 +408969.220}
SPL {X  -165.650, Y  +662.773, Z    +0.000, E1    +7.549, E3 +408969.142}
SPL {X  -165.650, Y  +656.581, Z    +0.000, E1   +13.870, E3 +408967.191}
SPL {X  -165.650, Y  +648.120, Z    +0.000, E1   +22.794, E3 +408966.422}
SPL {X  -165.650, Y  +632.103, Z    +0.000, E1   +42.949, E3 +408953.380}
SPL {X  -165.650, Y  +608.448, Z    +0.000, E1   +47.265, E3 +408979.820}
SPL {X  -165.650, Y  +595.526, Z    +0.000, E1   +48.856, E3 +408993.678}
SPL {X  -165.650, Y  +568.828, Z    +0.000, E1   +48.639, E3 +409036.231}
ENDSPLINE

SPLINE
SPL {X  -165.650, Y  +587.144, Z    +0.000, E1   +39.840, E3 +409050.264}
ENDSPLINE

SPLINE
SPL {X  -165.650, Y  +582.480, Z    +0.000, E1   +38.929, E3 +409067.460}
SPL {X  -165.650, Y  +575.679, Z    +0.000, E1   +38.947, E3 +409084.535}
SPL {X  -165.650, Y  +569.616, Z    +0.000, E1   +38.966, E3 +409099.693}
SPL {X  -165.650, Y  +564.364, Z    +0.000, E1   +38.909, E3 +409113.346}
SPL {X  -165.650, Y  +559.065, Z    +0.000, E1   +38.883, E3 +409126.924}
SPL {X  -165.650, Y  +552.770, Z    +0.000, E1   +38.963, E3 +409142.484}
SPL {X  -165.650, Y  +546.277, Z    +0.000, E1   +38.910, E3 +409159.226}
SPL {X  -165.650, Y  +540.151, Z    +0.000, E1   +38.996, E3 +409174.156}
SPL {X  -165.650, Y  +534.008, Z    +0.000, E1   +38.962, E3 +409189.998}
SPL {X  -165.650, Y  +528.320, Z    +0.000, E1   +38.809, E3 +409205.234}
SPL {X  -165.650, Y  +522.377, Z    +0.000, E1   +38.974, E3 +409219.354}
ENDSPLINE

SPLINE
SPL {X  -165.650, Y  +539.854, Z    +0.000, E1   +28.090, E3 +409235.971}
ENDSPLINE

SPLINE
SPL {X  -165.650, Y  +534.443, Z    +0.000, E1   +28.969, E3 +409250.022}
SPL {X  -165.650, Y  +530.452, Z    +0.000, E1   +29.664, E3 +409259.755}
SPL {X  -165.650, Y  +525.298, Z    +0.000, E1   +30.602, E3 +409271.566}
SPL {X  -165.650, Y  +518.290, Z    +0.000, E1   +31.783, E3 +409287.458}
SPL {X  -165.650, Y  +512.706, Z    +0.000, E1   +32.573, E3 +409300.292}
SPL {X  -165.650, Y  +507.785, Z    +0.000, E1   +33.438, E3 +409310.230}
SPL {X  -165.650, Y  +501.257, Z    +0.000, E1   +34.478, E3 +409323.469}
SPL {X  -165.650, Y  +493.800, Z    +0.000, E1   +35.486, E3 +409338.957}
SPL {X  -165.650, Y  +485.583, Z    +0.000, E1   +36.670, E3 +409354.681}
SPL {X  -165.650, Y  +477.375, Z    +0.000, E1   +37.747, E3 +409370.199}
SPL {X  -165.650, Y  +469.901, Z    +0.000, E1   +38.767, E3 +409383.331}
SPL {X  -165.650, Y  +465.276, Z    +0.000, E1   +39.067, E3 +409393.208}
SPL {X  -165.650, Y  +461.010, Z    +0.000, E1   +39.362, E3 +409402.171}
SPL {X  -165.650, Y  +457.119, Z    +0.000, E1   +39.087, E3 +409413.547}
SPL {X  -165.650, Y  +452.884, Z    +0.000, E1   +39.185, E3 +409423.595}
SPL {X  -165.650, Y  +449.593, Z    +0.000, E1   +38.852, E3 +409433.890}
SPL {X  -165.650, Y  +445.147, Z    +0.000, E1   +39.088, E3 +409443.712}
SPL {X  -165.650, Y  +439.751, Z    +0.000, E1   +39.254, E3 +409456.329}
SPL {X  -165.650, Y  +435.510, Z    +0.000, E1   +39.051, E3 +409468.141}
SPL {X  -165.650, Y  +430.832, Z    +0.000, E1   +39.105, E3 +409479.597}
SPL {X  -165.650, Y  +426.072, Z    +0.000, E1   +39.194, E3 +409491.020}
SPL {X  -165.650, Y  +422.372, Z    +0.000, E1   +38.952, E3 +409501.756}
SPL {X  -165.650, Y  +416.355, Z    +0.000, E1   +39.151, E3 +409515.916}
SPL {X  -165.650, Y  +408.927, Z    +0.000, E1   +39.115, E3 +409534.875}
SPL {X  -165.650, Y  +402.767, Z    +0.000, E1   +39.122, E3 +409550.136}
SPL {X  -165.650, Y  +398.352, Z    +0.000, E1   +39.113, E3 +409561.289}
SPL {X  -165.650, Y  +393.915, Z    +0.000, E1   +39.126, E3 +409572.366}
SPL {X  -165.650, Y  +389.523, Z    +0.000, E1   +39.115, E3 +409583.476}
SPL {X  -165.650, Y  +384.404, Z    +0.000, E1   +39.147, E3 +409596.212}
SPL {X  -165.650, Y  +378.675, Z    +0.000, E1   +39.090, E3 +409611.020}
SPL {X  -165.597, Y  +374.311, Z    +0.000, E1   +39.013, E3 +409622.306}
SPL {X  -165.438, Y  +370.129, Z    +0.000, E1   +39.090, E3 +409632.484}
SPL {X  -165.143, Y  +365.555, Z    +0.000, E1   +39.161, E3 +409643.456}
SPL {X  -164.909, Y  +362.853, Z    +0.000, E1   +38.709, E3 +409653.003}
SPL {X  -164.359, Y  +357.858, Z    +0.000, E1   +39.066, E3 +409663.465}
SPL {X  -163.818, Y  +353.935, Z    +0.000, E1   +38.811, E3 +409674.860}
SPL {X  -163.055, Y  +349.296, Z    +0.000, E1   +38.669, E3 +409687.365}
SPL {X  -162.319, Y  +345.445, Z    +0.000, E1   +38.490, E3 +409698.060}
SPL {X  -161.279, Y  +340.696, Z    +0.000, E1   +38.442, E3 +409710.388}
SPL {X  -160.251, Y  +336.552, Z    +0.000, E1   +38.166, E3 +409722.254}
SPL {X  -153.716, Y  +316.763, Z    +0.000, E1   +45.637, E3 +409724.872}
SPL {X  -149.011, Y  +306.142, Z    +0.000, E1   +47.422, E3 +409734.904}
SPL {X  -146.894, Y  +301.936, Z    +0.000, E1   +40.559, E3 +409803.141}
ENDSPLINE

SPLINE
SPL {X  -154.092, Y  +317.709, Z    +0.000, E1   +32.342, E3 +409872.266}
SPL {X  -161.950, Y  +343.684, Z    +0.000, E1   +21.785, E3 +409849.105}
SPL {X  -164.623, Y  +360.087, Z    +0.000, E1   +13.426, E3 +409857.756}
SPL {X  -165.588, Y  +373.983, Z    +0.000, E1    +5.738, E3 +409850.532}
SPL {X  -165.650, Y  +380.761, Z    +0.000, E1    +1.351, E3 +409852.257}
SPL {X  -165.650, Y  +386.484, Z    +0.000, E1    -2.972, E3 +409850.263}
SPL {X  -165.650, Y  +391.786, Z    +0.000, E1    -7.566, E3 +409852.659}
SPL {X  -165.650, Y  +395.964, Z    +0.000, E1   -11.741, E3 +409851.383}
SPL {X  -165.650, Y  +404.146, Z    +0.000, E1   -20.514, E3 +409847.048}
SPL {X  -165.650, Y  +416.920, Z    +0.000, E1   -34.832, E3 +409841.011}
SPL {X  -165.650, Y  +445.455, Z    +0.000, E1   -46.044, E3 +409863.101}
SPL {X  -165.650, Y  +459.839, Z    +0.000, E1   -48.128, E3 +409878.167}
SPL {X  -165.650, Y  +484.108, Z    +0.000, E1   -48.531, E3 +409915.159}
ENDSPLINE

SPLINE
SPL {X  -165.650, Y  +464.452, Z    +0.000, E1   -38.833, E3 +409930.220}
ENDSPLINE

SPLINE
SPL {X  -165.650, Y  +467.011, Z    +0.000, E1   -37.866, E3 +409942.644}
SPL {X  -165.650, Y  +471.256, Z    +0.000, E1   -37.789, E3 +409954.297}
SPL {X  -165.650, Y  +477.269, Z    +0.000, E1   -37.921, E3 +409969.514}
SPL {X  -165.650, Y  +483.881, Z    +0.000, E1   -37.934, E3 +409986.706}
SPL {X  -165.650, Y  +489.657, Z    +0.000, E1   -37.855, E3 +410002.367}
SPL {X  -165.650, Y  +496.067, Z    +0.000, E1   -37.879, E3 +410019.156}
SPL {X  -165.650, Y  +502.007, Z    +0.000, E1   -37.899, E3 +410034.538}
SPL {X  -165.650, Y  +506.838, Z    +0.000, E1   -38.018, E3 +410046.435}
SPL {X  -165.650, Y  +510.962, Z    +0.000, E1   -37.876, E3 +410058.149}
SPL {X  -165.650, Y  +513.924, Z    +0.000, E1   -37.557, E3 +410067.816}
SPL {X  -165.650, Y  +519.541, Z    +0.000, E1   -37.994, E3 +410080.151}
SPL {X  -165.650, Y  +524.168, Z    +0.000, E1   -37.816, E3 +410093.206}
SPL {X  -165.650, Y  +528.532, Z    +0.000, E1   -37.895, E3 +410104.272}
SPL {X  -165.650, Y  +532.864, Z    +0.000, E1   -37.846, E3 +410115.914}
SPL {X  -165.650, Y  +537.279, Z    +0.000, E1   -37.980, E3 +410126.737}
SPL {X  -165.650, Y  +540.651, Z    +0.000, E1   -37.651, E3 +410137.539}
SPL {X  -165.650, Y  +545.726, Z    +0.000, E1   -37.963, E3 +410149.104}
SPL {X  -165.650, Y  +550.427, Z    +0.000, E1   -37.784, E3 +410162.522}
SPL {X  -165.650, Y  +556.372, Z    +0.000, E1   -37.998, E3 +410176.918}
SPL {X  -165.650, Y  +561.478, Z    +0.000, E1   -37.846, E3 +410191.166}
SPL {X  -165.650, Y  +566.625, Z    +0.000, E1   -37.932, E3 +410204.195}
SPL {X  -165.650, Y  +571.305, Z    +0.000, E1   -37.718, E3 +410217.832}
SPL {X  -165.650, Y  +577.754, Z    +0.000, E1   -38.006, E3 +410233.124}
SPL {X  -165.650, Y  +583.042, Z    +0.000, E1   -37.879, E3 +410247.667}
SPL {X  -165.650, Y  +587.643, Z    +0.000, E1   -37.879, E3 +410259.745}
SPL {X  -165.650, Y  +592.833, Z    +0.000, E1   -37.896, E3 +410273.394}
SPL {X  -165.650, Y  +597.119, Z    +0.000, E1   -37.642, E3 +410286.123}
SPL {X  -165.650, Y  +602.808, Z    +0.000, E1   -37.983, E3 +410299.129}
SPL {X  -165.650, Y  +607.937, Z    +0.000, E1   -37.862, E3 +410313.291}
SPL {X  -165.650, Y  +614.056, Z    +0.000, E1   -37.933, E3 +410329.061}
SPL {X  -165.650, Y  +619.142, Z    +0.000, E1   -37.954, E3 +410342.080}
SPL {X  -165.650, Y  +622.884, Z    +0.000, E1   -37.770, E3 +410353.123}
SPL {X  -165.650, Y  +627.016, Z    +0.000, E1   -37.897, E3 +410363.161}
SPL {X  -165.650, Y  +630.421, Z    +0.000, E1   -38.020, E3 +410371.324}
SPL {X  -165.650, Y  +633.686, Z    +0.000, E1   -37.760, E3 +410381.568}
SPL {X  -165.650, Y  +638.669, Z    +0.000, E1   -37.941, E3 +410393.574}
SPL {X  -165.650, Y  +643.208, Z    +0.000, E1   -37.786, E3 +410406.491}
SPL {X  -165.650, Y  +649.293, Z    +0.000, E1   -37.920, E3 +410421.781}
SPL {X  -165.650, Y  +654.711, Z    +0.000, E1   -37.888, E3 +410436.103}
SPL {X  -165.650, Y  +658.674, Z    +0.000, E1   -37.902, E3 +410446.371}
SPL {X  -165.650, Y  +661.754, Z    +0.000, E1   -37.878, E3 +410454.607}
SPL {X  -165.650, Y  +665.663, Z    +0.000, E1   -37.913, E3 +410464.708}
SPL {X  -165.650, Y  +669.913, Z    +0.000, E1   -37.905, E3 +410475.910}
SPL {X  -165.650, Y  +674.729, Z    +0.000, E1   -37.860, E3 +410488.920}
SPL {X  -165.591, Y  +679.928, Z    +0.000, E1   -37.818, E3 +410502.837}
SPL {X  -165.340, Y  +685.624, Z    +0.000, E1   -37.900, E3 +410517.372}
SPL {X  -165.010, Y  +690.051, Z    +0.000, E1   -37.675, E3 +410530.303}
SPL {X  -164.652, Y  +693.652, Z    +0.000, E1   -37.750, E3 +410539.233}
SPL {X  -164.143, Y  +697.797, Z    +0.000, E1   -37.636, E3 +410551.052}
SPL {X  -163.447, Y  +702.423, Z    +0.000, E1   -37.496, E3 +410563.861}
SPL {X  -162.809, Y  +706.049, Z    +0.000, E1   -37.384, E3 +410574.131}
SPL {X  -161.803, Y  +710.992, Z    +0.000, E1   -37.315, E3 +410587.596}
SPL {X  -160.993, Y  +714.501, Z    +0.000, E1   -36.839, E3 +410599.472}
SPL {X  -159.156, Y  +721.427, Z    +0.000, E1   -38.526, E3 +410607.550}
SPL {X  -144.831, Y  +755.898, Z    +0.000, E1   -42.981, E3 +410668.966}
ENDSPLINE

SPLINE
SPL {X  -153.047, Y  +738.876, Z    +0.000, E1   -33.363, E3 +410751.181}
SPL {X  -162.649, Y  +706.888, Z    +0.000, E1   -19.911, E3 +410740.543}
SPL {X  -165.011, Y  +690.033, Z    +0.000, E1   -11.292, E3 +410736.777}
SPL {X  -165.581, Y  +680.273, Z    +0.000, E1    -5.775, E3 +410732.576}
SPL {X  -165.650, Y  +674.660, Z    +0.000, E1    -2.196, E3 +410733.243}
SPL {X  -165.650, Y  +669.932, Z    +0.000, E1    +1.173, E3 +410731.819}
SPL {X  -165.650, Y  +665.412, Z    +0.000, E1    +4.953, E3 +410730.998}
SPL {X  -165.650, Y  +658.891, Z    +0.000, E1   +11.031, E3 +410731.309}
SPL {X  -165.650, Y  +649.186, Z    +0.000, E1   +20.530, E3 +410732.569}
SPL {X  -165.650, Y  +637.823, Z    +0.000, E1   +39.473, E3 +410712.165}
SPL {X  -165.650, Y  +613.283, Z    +0.000, E1   +49.826, E3 +410727.732}
SPL {X  -165.650, Y  +609.693, Z    +0.000, E1   +42.113, E3 +410755.866}
SPL {X  -165.650, Y  +571.563, Z    +0.000, E1   +48.716, E3 +410794.184}
SPL {X  -165.650, Y  +570.963, Z    +0.000, E1   +46.818, E3 +410805.712}
ENDSPLINE

SPLINE
SPL {X  -165.650, Y  +586.477, Z    +0.000, E1   +39.172, E3 +410817.220}
ENDSPLINE

SPLINE
SPL {X  -165.650, Y  +581.917, Z    +0.000, E1   +39.019, E3 +410829.622}
SPL {X  -165.650, Y  +577.218, Z    +0.000, E1   +38.911, E3 +410842.162}
SPL {X  -165.650, Y  +571.720, Z    +0.000, E1   +39.004, E3 +410855.554}
SPL {X  -165.650, Y  +565.656, Z    +0.000, E1   +39.042, E3 +410870.663}
SPL {X  -165.650, Y  +560.333, Z    +0.000, E1   +38.995, E3 +410884.292}
SPL {X  -165.650, Y  +554.558, Z    +0.000, E1   +39.065, E3 +410898.580}
SPL {X  -165.650, Y  +548.147, Z    +0.000, E1   +39.104, E3 +410914.437}
SPL {X  -165.650, Y  +526.098, Z    +0.000, E1   +45.792, E3 +410924.256}
SPL {X  -165.650, Y  +510.223, Z    +0.000, E1   +49.521, E3 +410931.653}
SPL {X  -165.650, Y  +506.429, Z    +0.000, E1   +48.913, E3 +410942.066}
SPL {X  -165.650, Y  +501.394, Z    +0.000, E1   +48.110, E3 +410956.045}
SPL {X  -165.650, Y  +497.138, Z    +0.000, E1   +47.280, E3 +410968.741}
SPL {X  -165.650, Y  +493.273, Z    +0.000, E1   +46.518, E3 +410980.722}
SPL {X  -165.650, Y  +489.140, Z    +0.000, E1   +45.675, E3 +410993.849}
SPL {X  -165.650, Y  +485.420, Z    +0.000, E1   +44.711, E3 +411007.068}
SPL {X  -165.650, Y  +480.756, Z    +0.000, E1   +43.779, E3 +411022.546}
SPL {X  -165.650, Y  +475.837, Z    +0.000, E1   +42.787, E3 +411039.007}
SPL {X  -165.650, Y  +472.413, Z    +0.000, E1   +41.852, E3 +411052.121}
SPL {X  -165.650, Y  +469.721, Z    +0.000, E1   +41.361, E3 +411061.148}
SPL {X  -165.650, Y  +467.130, Z    +0.000, E1   +40.624, E3 +411071.830}
SPL {X  -165.650, Y  +463.869, Z    +0.000, E1   +39.839, E3 +411084.298}
SPL {X  -165.650, Y  +462.171, Z    +0.000, E1   +38.860, E3 +411094.477}
SPL {X  -165.650, Y  +457.119, Z    +0.000, E1   +39.087, E3 +411105.855}
SPL {X  -165.650, Y  +452.884, Z    +0.000, E1   +39.185, E3 +411115.903}
SPL {X  -165.650, Y  +449.593, Z    +0.000, E1   +38.852, E3 +411126.198}
SPL {X  -165.650, Y  +445.147, Z    +0.000, E1   +39.088, E3 +411136.020}
SPL {X  -165.650, Y  +439.751, Z    +0.000, E1   +39.254, E3 +411148.637}
SPL {X  -165.650, Y  +435.510, Z    +0.000, E1   +39.051, E3 +411160.448}
SPL {X  -165.650, Y  +430.832, Z    +0.000, E1   +39.105, E3 +411171.905}
SPL {X  -165.650, Y  +426.072, Z    +0.000, E1   +39.194, E3 +411183.328}
SPL {X  -165.650, Y  +422.372, Z    +0.000, E1   +38.952, E3 +411194.064}
SPL {X  -165.650, Y  +417.591, Z    +0.000, E1   +39.157, E3 +411204.917}
SPL {X  -165.650, Y  +412.842, Z    +0.000, E1   +39.072, E3 +411217.416}
SPL {X  -165.650, Y  +407.612, Z    +0.000, E1   +39.068, E3 +411230.588}
SPL {X  -165.650, Y  +402.767, Z    +0.000, E1   +39.122, E3 +411242.444}
SPL {X  -165.650, Y  +398.352, Z    +0.000, E1   +39.113, E3 +411253.597}
SPL {X  -165.650, Y  +393.915, Z    +0.000, E1   +39.126, E3 +411264.674}
SPL {X  -165.650, Y  +389.523, Z    +0.000, E1   +39.115, E3 +411275.784}
SPL {X  -165.650, Y  +384.404, Z    +0.000, E1   +39.147, E3 +411288.520}
SPL {X  -165.650, Y  +380.058, Z    +0.000, E1   +39.073, E3 +411299.807}
SPL {X  -165.624, Y  +375.547, Z    +0.000, E1   +39.047, E3 +411311.406}
SPL {X  -165.438, Y  +370.129, Z    +0.000, E1   +39.090, E3 +411324.791}
SPL {X  -165.143, Y  +365.555, Z    +0.000, E1   +39.161, E3 +411335.764}
SPL {X  -164.909, Y  +362.853, Z    +0.000, E1   +38.709, E3 +411345.310}
SPL {X  -164.359, Y  +357.858, Z    +0.000, E1   +39.066, E3 +411355.773}
SPL {X  -163.818, Y  +353.935, Z    +0.000, E1   +38.811, E3 +411367.167}
SPL {X  -163.055, Y  +349.296, Z    +0.000, E1   +38.669, E3 +411379.673}
SPL {X  -162.021, Y  +344.016, Z    +0.000, E1   +38.517, E3 +411393.962}
SPL {X  -160.588, Y  +337.861, Z    +0.000, E1   +38.304, E3 +411410.676}
SPL {X  -151.400, Y  +311.284, Z    +0.000, E1   +46.597, E3 +411422.285}
SPL {X  -146.894, Y  +301.936, Z    +0.000, E1   +40.559, E3 +411495.449}
ENDSPLINE

SPLINE
SPL {X  -154.092, Y  +317.709, Z    +0.000, E1   +32.342, E3 +411564.573}
SPL {X  -161.950, Y  +343.684, Z    +0.000, E1   +21.785, E3 +411541.413}
SPL {X  -164.623, Y  +360.087, Z    +0.000, E1   +13.426, E3 +411550.063}
SPL {X  -165.588, Y  +373.983, Z    +0.000, E1    +5.738, E3 +411542.840}
SPL {X  -165.650, Y  +380.761, Z    +0.000, E1    +1.351, E3 +411544.564}
SPL {X  -165.650, Y  +385.186, Z    +0.000, E1    -1.985, E3 +411543.049}
SPL {X  -165.650, Y  +387.866, Z    +0.000, E1    -4.228, E3 +411542.062}
SPL {X  -165.650, Y  +391.786, Z    +0.000, E1    -7.566, E3 +411544.966}
SPL {X  -165.650, Y  +399.284, Z    +0.000, E1   -15.403, E3 +411540.151}
SPL {X  -165.650, Y  +409.824, Z    +0.000, E1   -26.455, E3 +411538.031}
SPL {X  -165.650, Y  +437.337, Z    +0.000, E1   -46.817, E3 +411540.666}
SPL {X  -165.650, Y  +450.640, Z    +0.000, E1   -46.274, E3 +411562.688}
SPL {X  -165.650, Y  +484.108, Z    +0.000, E1   -48.531, E3 +411607.467}
ENDSPLINE

SPLINE
SPL {X  -165.650, Y  +464.452, Z    +0.000, E1   -38.833, E3 +411622.527}
ENDSPLINE

SPLINE
SPL {X  -165.650, Y  +467.011, Z    +0.000, E1   -37.866, E3 +411634.951}
SPL {X  -165.650, Y  +471.256, Z    +0.000, E1   -37.789, E3 +411646.605}
SPL {X  -165.650, Y  +475.981, Z    +0.000, E1   -37.909, E3 +411658.328}
SPL {X  -165.650, Y  +481.142, Z    +0.000, E1   -37.875, E3 +411672.148}
SPL {X  -165.650, Y  +487.016, Z    +0.000, E1   -37.964, E3 +411687.053}
SPL {X  -165.650, Y  +490.835, Z    +0.000, E1   -37.708, E3 +411698.501}
SPL {X  -165.650, Y  +496.067, Z    +0.000, E1   -37.879, E3 +411711.464}
SPL {X  -165.650, Y  +502.007, Z    +0.000, E1   -37.899, E3 +411726.846}
SPL {X  -165.650, Y  +506.838, Z    +0.000, E1   -38.018, E3 +411738.743}
SPL {X  -165.650, Y  +510.962, Z    +0.000, E1   -37.876, E3 +411750.457}
SPL {X  -165.650, Y  +513.924, Z    +0.000, E1   -37.557, E3 +411760.124}
SPL {X  -165.650, Y  +519.541, Z    +0.000, E1   -37.994, E3 +411772.459}
SPL {X  -165.650, Y  +524.168, Z    +0.000, E1   -37.816, E3 +411785.514}
SPL {X  -165.650, Y  +528.532, Z    +0.000, E1   -37.895, E3 +411796.580}
SPL {X  -165.650, Y  +532.864, Z    +0.000, E1   -37.846, E3 +411808.222}
SPL {X  -165.650, Y  +537.279, Z    +0.000, E1   -37.980, E3 +411819.044}
SPL {X  -165.650, Y  +540.651, Z    +0.000, E1   -37.651, E3 +411829.847}
SPL {X  -165.650, Y  +545.726, Z    +0.000, E1   -37.963, E3 +411841.412}
SPL {X  -165.650, Y  +550.427, Z    +0.000, E1   -37.784, E3 +411854.830}
SPL {X  -165.650, Y  +554.659, Z    +0.000, E1   -37.927, E3 +411865.014}
SPL {X  -165.650, Y  +557.856, Z    +0.000, E1   -37.998, E3 +411872.964}
SPL {X  -165.650, Y  +562.748, Z    +0.000, E1   -37.890, E3 +411886.707}
SPL {X  -165.650, Y  +567.848, Z    +0.000, E1   -37.954, E3 +411899.479}
SPL {X  -165.650, Y  +571.305, Z    +0.000, E1   -37.718, E3 +411910.140}
SPL {X  -165.650, Y  +577.754, Z    +0.000, E1   -38.006, E3 +411925.432}
SPL {X  -165.650, Y  +583.042, Z    +0.000, E1   -37.879, E3 +411939.975}
SPL {X  -165.650, Y  +587.643, Z    +0.000, E1   -37.879, E3 +411952.053}
SPL {X  -165.650, Y  +592.833, Z    +0.000, E1   -37.896, E3 +411965.702}
SPL {X  -165.650, Y  +599.187, Z    +0.000, E1   -37.841, E3 +411982.840}
SPL {X  -165.650, Y  +604.276, Z    +0.000, E1   -37.917, E3 +411995.527}
SPL {X  -165.650, Y  +607.937, Z    +0.000, E1   -37.862, E3 +412005.598}
SPL {X  -165.650, Y  +612.863, Z    +0.000, E1   -37.857, E3 +412018.571}
SPL {X  -165.650, Y  +618.208, Z    +0.000, E1   -37.992, E3 +412031.813}
SPL {X  -165.650, Y  +622.884, Z    +0.000, E1   -37.770, E3 +412045.430}
SPL {X  -165.650, Y  +628.759, Z    +0.000, E1   -37.993, E3 +412059.600}
SPL {X  -165.650, Y  +633.686, Z    +0.000, E1   -37.760, E3 +412073.876}
SPL {X  -165.650, Y  +638.669, Z    +0.000, E1   -37.941, E3 +412085.882}
SPL {X  -165.650, Y  +644.441, Z    +0.000, E1   -37.838, E3 +412101.897}
SPL {X  -165.650, Y  +650.450, Z    +0.000, E1   -37.924, E3 +412116.976}
SPL {X  -165.650, Y  +654.711, Z    +0.000, E1   -37.888, E3 +412128.410}
SPL {X  -165.650, Y  +660.285, Z    +0.000, E1   -37.928, E3 +412142.929}
SPL {X  -165.650, Y  +665.663, Z    +0.000, E1   -37.913, E3 +412157.016}
SPL {X  -165.650, Y  +669.913, Z    +0.000, E1   -37.905, E3 +412168.218}
SPL {X  -165.650, Y  +674.729, Z    +0.000, E1   -37.860, E3 +412181.227}
SPL {X  -165.591, Y  +679.928, Z    +0.000, E1   -37.818, E3 +412195.145}
SPL {X  -165.340, Y  +685.624, Z    +0.000, E1   -37.900, E3 +412209.679}
SPL {X  -164.889, Y  +691.361, Z    +0.000, E1   -37.742, E3 +412225.797}
SPL {X  -164.246, Y  +697.018, Z    +0.000, E1   -37.690, E3 +412240.840}
SPL {X  -163.617, Y  +701.375, Z    +0.000, E1   -37.486, E3 +412253.567}
SPL {X  -162.809, Y  +706.049, Z    +0.000, E1   -37.384, E3 +412266.439}
SPL {X  -162.124, Y  +709.497, Z    +0.000, E1   -37.325, E3 +412275.761}
SPL {X  -161.242, Y  +713.462, Z    +0.000, E1   -37.074, E3 +412287.882}
SPL {X  -159.156, Y  +721.427, Z    +0.000, E1   -38.526, E3 +412299.858}
SPL {X  -144.831, Y  +755.898, Z    +0.000, E1   -42.981, E3 +412361.274}
ENDSPLINE

SPLINE
SPL {X  -153.047, Y  +738.876, Z    +0.000, E1   -33.363, E3 +412443.489}
SPL {X  -162.649, Y  +706.888, Z    +0.000, E1   -19.911, E3 +412432.851}
SPL {X  -165.011, Y  +690.033, Z    +0.000, E1   -11.292, E3 +412429.085}
SPL {X  -165.581, Y  +680.273, Z    +0.000, E1    -5.775, E3 +412424.883}
SPL {X  -165.650, Y  +674.660, Z    +0.000, E1    -2.196, E3 +412425.550}
SPL {X  -165.650, Y  +669.932, Z    +0.000, E1    +1.173, E3 +412424.126}
SPL {X  -165.650, Y  +665.412, Z    +0.000, E1    +4.953, E3 +412423.306}
SPL {X  -165.650, Y  +658.891, Z    +0.000, E1   +11.031, E3 +412423.617}
SPL {X  -165.650, Y  +649.186, Z    +0.000, E1   +20.530, E3 +412424.877}
SPL {X  -165.650, Y  +637.823, Z    +0.000, E1   +39.473, E3 +412404.473}
SPL {X  -165.650, Y  +613.283, Z    +0.000, E1   +49.826, E3 +412420.040}
SPL {X  -165.650, Y  +609.693, Z    +0.000, E1   +42.113, E3 +412448.174}
SPL {X  -165.650, Y  +571.120, Z    +0.000, E1   +47.704, E3 +412492.983}
ENDSPLINE

SPLINE
SPL {X  -165.650, Y  +586.477, Z    +0.000, E1   +39.172, E3 +412509.527}
ENDSPLINE

SPLINE
SPL {X  -165.650, Y  +581.917, Z    +0.000, E1   +39.019, E3 +412521.930}
SPL {X  -165.650, Y  +577.218, Z    +0.000, E1   +38.911, E3 +412534.470}
SPL {X  -165.650, Y  +572.890, Z    +0.000, E1   +39.033, E3 +412544.608}
SPL {X  -165.650, Y  +569.005, Z    +0.000, E1   +38.999, E3 +412554.698}
SPL {X  -165.650, Y  +564.604, Z    +0.000, E1   +38.986, E3 +412565.834}
SPL {X  -165.650, Y  +560.333, Z    +0.000, E1   +38.995, E3 +412576.599}
SPL {X  -165.650, Y  +556.690, Z    +0.000, E1   +39.061, E3 +412585.318}
SPL {X  -165.650, Y  +552.186, Z    +0.000, E1   +39.063, E3 +412596.836}
SPL {X  -165.650, Y  +547.091, Z    +0.000, E1   +39.070, E3 +412609.496}
SPL {X  -165.650, Y  +526.098, Z    +0.000, E1   +45.792, E3 +412616.563}
SPL {X  -165.650, Y  +510.223, Z    +0.000, E1   +49.521, E3 +412623.960}
SPL {X  -165.650, Y  +506.429, Z    +0.000, E1   +48.913, E3 +412634.373}
SPL {X  -165.650, Y  +501.394, Z    +0.000, E1   +48.110, E3 +412648.352}
SPL {X  -165.650, Y  +497.138, Z    +0.000, E1   +47.280, E3 +412661.048}
SPL {X  -165.650, Y  +493.273, Z    +0.000, E1   +46.518, E3 +412673.029}
SPL {X  -165.650, Y  +489.140, Z    +0.000, E1   +45.675, E3 +412686.157}
SPL {X  -165.650, Y  +485.420, Z    +0.000, E1   +44.711, E3 +412699.376}
SPL {X  -165.650, Y  +480.756, Z    +0.000, E1   +43.779, E3 +412714.854}
SPL {X  -165.650, Y  +475.837, Z    +0.000, E1   +42.787, E3 +412731.314}
SPL {X  -165.650, Y  +472.413, Z    +0.000, E1   +41.852, E3 +412744.429}
SPL {X  -165.650, Y  +468.649, Z    +0.000, E1   +41.090, E3 +412757.793}
SPL {X  -165.650, Y  +465.438, Z    +0.000, E1   +39.745, E3 +412773.589}
SPL {X  -165.650, Y  +461.167, Z    +0.000, E1   +39.270, E3 +412786.924}
SPL {X  -165.650, Y  +457.119, Z    +0.000, E1   +39.087, E3 +412798.163}
SPL {X  -165.650, Y  +452.884, Z    +0.000, E1   +39.185, E3 +412808.210}
SPL {X  -165.650, Y  +449.593, Z    +0.000, E1   +38.852, E3 +412818.505}
SPL {X  -165.650, Y  +445.147, Z    +0.000, E1   +39.088, E3 +412828.328}
SPL {X  -165.650, Y  +439.751, Z    +0.000, E1   +39.254, E3 +412840.945}
SPL {X  -165.650, Y  +435.510, Z    +0.000, E1   +39.051, E3 +412852.756}
SPL {X  -165.650, Y  +430.832, Z    +0.000, E1   +39.105, E3 +412864.213}
SPL {X  -165.650, Y  +426.072, Z    +0.000, E1   +39.194, E3 +412875.636}
SPL {X  -165.650, Y  +422.372, Z    +0.000, E1   +38.952, E3 +412886.371}
SPL {X  -165.650, Y  +416.355, Z    +0.000, E1   +39.151, E3 +412900.531}
SPL {X  -165.650, Y  +408.927, Z    +0.000, E1   +39.115, E3 +412919.490}
SPL {X  -165.650, Y  +402.767, Z    +0.000, E1   +39.122, E3 +412934.751}
SPL {X  -165.650, Y  +398.352, Z    +0.000, E1   +39.113, E3 +412945.904}
SPL {X  -165.650, Y  +393.915, Z    +0.000, E1   +39.126, E3 +412956.981}
SPL {X  -165.650, Y  +389.523, Z    +0.000, E1   +39.115, E3 +412968.091}
SPL {X  -165.650, Y  +384.404, Z    +0.000, E1   +39.147, E3 +412980.827}
SPL {X  -165.650, Y  +378.675, Z    +0.000, E1   +39.090, E3 +412995.636}
SPL {X  -165.597, Y  +374.311, Z    +0.000, E1   +39.013, E3 +413006.921}
SPL {X  -165.438, Y  +370.129, Z    +0.000, E1   +39.090, E3 +413017.099}
SPL {X  -165.143, Y  +365.555, Z    +0.000, E1   +39.161, E3 +413028.072}
SPL {X  -164.909, Y  +362.853, Z    +0.000, E1   +38.709, E3 +413037.618}
SPL {X  -164.359, Y  +357.858, Z    +0.000, E1   +39.066, E3 +413048.081}
SPL {X  -163.818, Y  +353.935, Z    +0.000, E1   +38.811, E3 +413059.475}
SPL {X  -163.055, Y  +349.296, Z    +0.000, E1   +38.669, E3 +413071.980}
SPL {X  -162.319, Y  +345.445, Z    +0.000, E1   +38.490, E3 +413082.676}
SPL {X  -161.279, Y  +340.696, Z    +0.000, E1   +38.442, E3 +413095.003}
SPL {X  -160.251, Y  +336.552, Z    +0.000, E1   +38.166, E3 +413106.869}
SPL {X  -151.400, Y  +311.284, Z    +0.000, E1   +46.597, E3 +413114.592}
SPL {X  -146.894, Y  +301.936, Z    +0.000, E1   +40.559, E3 +413187.757}
ENDSPLINE

SPLINE
SPL {X  -154.092, Y  +317.709, Z    +0.000, E1   +32.342, E3 +413256.881}
SPL {X  -161.950, Y  +343.684, Z    +0.000, E1   +21.785, E3 +413233.720}
SPL {X  -164.623, Y  +360.087, Z    +0.000, E1   +13.426, E3 +413242.371}
SPL {X  -165.588, Y  +373.983, Z    +0.000, E1    +5.738, E3 +413235.148}
SPL {X  -165.650, Y  +380.761, Z    +0.000, E1    +1.351, E3 +413236.872}
SPL {X  -165.650, Y  +386.484, Z    +0.000, E1    -2.972, E3 +413234.879}
SPL {X  -165.650, Y  +392.905, Z    +0.000, E1    -8.557, E3 +413236.933}
SPL {X  -165.650, Y  +404.146, Z    +0.000, E1   -20.514, E3 +413231.663}
SPL {X  -165.650, Y  +416.920, Z    +0.000, E1   -34.832, E3 +413225.626}
SPL {X  -165.650, Y  +445.455, Z    +0.000, E1   -46.044, E3 +413247.717}
SPL {X  -165.650, Y  +459.839, Z    +0.000, E1   -48.128, E3 +413262.783}
SPL {X  -165.650, Y  +484.108, Z    +0.000, E1   -48.531, E3 +413299.774}
ENDSPLINE

SPLINE
SPL {X  -165.650, Y  +464.452, Z    +0.000, E1   -38.833, E3 +413314.835}
ENDSPLINE

SPLINE
SPL {X  -165.650, Y  +467.011, Z    +0.000, E1   -37.866, E3 +413327.259}
SPL {X  -165.650, Y  +471.256, Z    +0.000, E1   -37.789, E3 +413338.913}
SPL {X  -165.650, Y  +475.981, Z    +0.000, E1   -37.909, E3 +413350.636}
SPL {X  -165.650, Y  +481.142, Z    +0.000, E1   -37.875, E3 +413364.456}
SPL {X  -165.650, Y  +487.016, Z    +0.000, E1   -37.964, E3 +413379.361}
SPL {X  -165.650, Y  +492.473, Z    +0.000, E1   -37.882, E3 +413394.158}
SPL {X  -165.650, Y  +496.967, Z    +0.000, E1   -37.731, E3 +413406.865}
SPL {X  -165.650, Y  +502.007, Z    +0.000, E1   -37.899, E3 +413419.154}
SPL {X  -165.650, Y  +507.602, Z    +0.000, E1   -37.863, E3 +413434.184}
SPL {X  -165.650, Y  +513.428, Z    +0.000, E1   -37.892, E3 +413449.249}
SPL {X  -165.650, Y  +519.541, Z    +0.000, E1   -37.994, E3 +413464.766}
SPL {X  -165.650, Y  +524.168, Z    +0.000, E1   -37.816, E3 +413477.822}
SPL {X  -165.650, Y  +528.532, Z    +0.000, E1   -37.895, E3 +413488.888}
SPL {X  -165.650, Y  +532.864, Z    +0.000, E1   -37.846, E3 +413500.529}
SPL {X  -165.650, Y  +537.279, Z    +0.000, E1   -37.980, E3 +413511.352}
SPL {X  -165.650, Y  +540.651, Z    +0.000, E1   -37.651, E3 +413522.154}
SPL {X  -165.650, Y  +545.726, Z    +0.000, E1   -37.963, E3 +413533.720}
SPL {X  -165.650, Y  +550.427, Z    +0.000, E1   -37.784, E3 +413547.138}
SPL {X  -165.650, Y  +556.372, Z    +0.000, E1   -37.998, E3 +413561.534}
SPL {X  -165.650, Y  +562.748, Z    +0.000, E1   -37.890, E3 +413579.014}
SPL {X  -165.650, Y  +567.848, Z    +0.000, E1   -37.954, E3 +413591.787}
SPL {X  -165.650, Y  +571.305, Z    +0.000, E1   -37.718, E3 +413602.448}
SPL {X  -165.650, Y  +577.754, Z    +0.000, E1   -38.006, E3 +413617.739}
SPL {X  -165.650, Y  +583.042, Z    +0.000, E1   -37.879, E3 +413632.283}
SPL {X  -165.650, Y  +588.969, Z    +0.000, E1   -37.907, E3 +413647.848}
SPL {X  -165.650, Y  +594.102, Z    +0.000, E1   -37.878, E3 +413661.317}
SPL {X  -165.650, Y  +597.119, Z    +0.000, E1   -37.642, E3 +413670.738}
SPL {X  -165.650, Y  +602.808, Z    +0.000, E1   -37.983, E3 +413683.744}
SPL {X  -165.650, Y  +607.937, Z    +0.000, E1   -37.862, E3 +413697.906}
SPL {X  -165.650, Y  +614.056, Z    +0.000, E1   -37.933, E3 +413713.677}
SPL {X  -165.650, Y  +619.142, Z    +0.000, E1   -37.954, E3 +413726.695}
SPL {X  -165.650, Y  +622.884, Z    +0.000, E1   -37.770, E3 +413737.738}
SPL {X  -165.650, Y  +628.759, Z    +0.000, E1   -37.993, E3 +413751.908}
SPL {X  -165.650, Y  +633.686, Z    +0.000, E1   -37.760, E3 +413766.183}
SPL {X  -165.650, Y  +639.918, Z    +0.000, E1   -37.892, E3 +413781.992}
SPL {X  -165.650, Y  +645.851, Z    +0.000, E1   -37.854, E3 +413797.644}
SPL {X  -165.650, Y  +650.450, Z    +0.000, E1   -37.924, E3 +413809.284}
SPL {X  -165.650, Y  +654.711, Z    +0.000, E1   -37.888, E3 +413820.718}
SPL {X  -165.650, Y  +658.674, Z    +0.000, E1   -37.902, E3 +413830.986}
SPL {X  -165.650, Y  +661.754, Z    +0.000, E1   -37.878, E3 +413839.222}
SPL {X  -165.650, Y  +665.663, Z    +0.000, E1   -37.913, E3 +413849.324}
SPL {X  -165.650, Y  +669.913, Z    +0.000, E1   -37.905, E3 +413860.526}
SPL {X  -165.650, Y  +674.729, Z    +0.000, E1   -37.860, E3 +413873.535}
SPL {X  -165.554, Y  +681.132, Z    +0.000, E1   -37.883, E3 +413890.370}
SPL {X  -165.277, Y  +686.615, Z    +0.000, E1   -37.853, E3 +413904.751}
SPL {X  -164.889, Y  +691.361, Z    +0.000, E1   -37.742, E3 +413918.105}
SPL {X  -164.246, Y  +697.018, Z    +0.000, E1   -37.690, E3 +413933.147}
SPL {X  -163.617, Y  +701.375, Z    +0.000, E1   -37.486, E3 +413945.875}
SPL {X  -162.809, Y  +706.049, Z    +0.000, E1   -37.384, E3 +413958.746}
SPL {X  -161.803, Y  +710.992, Z    +0.000, E1   -37.315, E3 +413972.211}
SPL {X  -160.993, Y  +714.501, Z    +0.000, E1   -36.839, E3 +413984.087}
SPL {X  -159.156, Y  +721.427, Z    +0.000, E1   -38.526, E3 +413992.166}
SPL {X  -144.831, Y  +755.898, Z    +0.000, E1   -42.981, E3 +414053.582}
ENDSPLINE

SPLINE
SPL {X  -153.047, Y  +738.876, Z    +0.000, E1   -33.363, E3 +414135.796}
SPL {X  -162.649, Y  +706.888, Z    +0.000, E1   -19.911, E3 +414125.158}
SPL {X  -165.011, Y  +690.033, Z    +0.000, E1   -11.292, E3 +414121.393}
SPL {X  -165.581, Y  +680.273, Z    +0.000, E1    -5.775, E3 +414117.191}
SPL {X  -165.650, Y  +674.660, Z    +0.000, E1    -2.196, E3 +414117.858}
SPL {X  -165.650, Y  +669.932, Z    +0.000, E1    +1.173, E3 +414116.434}
SPL {X  -165.650, Y  +665.412, Z    +0.000, E1    +4.953, E3 +414115.614}
SPL {X  -165.650, Y  +660.335, Z    +0.000, E1    +9.682, E3 +414116.131}
SPL {X  -165.650, Y  +650.970, Z    +0.000, E1   +18.783, E3 +414116.679}
SPL {X  -165.650, Y  +637.823, Z    +0.000, E1   +39.473, E3 +414096.780}
SPL {X  -165.650, Y  +614.460, Z    +0.000, E1   +51.116, E3 +414107.649}
SPL {X  -165.650, Y  +609.746, Z    +0.000, E1   +42.762, E3 +414138.307}
SPL {X  -165.650, Y  +571.120, Z    +0.000, E1   +47.704, E3 +414185.291}
ENDSPLINE

SPLINE
SPL {X  -165.650, Y  +586.477, Z    +0.000, E1   +39.172, E3 +414201.835}
ENDSPLINE

SPLINE
SPL {X  -165.650, Y  +581.917, Z    +0.000, E1   +39.019, E3 +414214.237}
SPL {X  -165.650, Y  +577.218, Z    +0.000, E1   +38.911, E3 +414226.778}
SPL {X  -165.650, Y  +572.890, Z    +0.000, E1   +39.033, E3 +414236.915}
SPL {X  -165.650, Y  +569.005, Z    +0.000, E1   +38.999, E3 +414247.006}
SPL {X  -165.650, Y  +564.604, Z    +0.000, E1   +38.986, E3 +414258.141}
SPL {X  -165.650, Y  +558.931, Z    +0.000, E1   +39.059, E3 +414272.209}
SPL {X  -165.650, Y  +553.380, Z    +0.000, E1   +39.004, E3 +414286.372}
SPL {X  -165.650, Y  +548.147, Z    +0.000, E1   +39.104, E3 +414299.052}
SPL {X  -165.650, Y  +526.098, Z    +0.000, E1   +45.792, E3 +414308.871}
SPL {X  -165.650, Y  +510.223, Z    +0.000, E1   +49.521, E3 +414316.268}
SPL {X  -165.650, Y  +506.429, Z    +0.000, E1   +48.913, E3 +414326.681}
SPL {X  -165.650, Y  +501.394, Z    +0.000, E1   +48.110, E3 +414340.660}
SPL {X  -165.650, Y  +497.138, Z    +0.000, E1   +47.280, E3 +414353.356}
SPL {X  -165.650, Y  +493.273, Z    +0.000, E1   +46.518, E3 +414365.337}
SPL {X  -165.650, Y  +490.148, Z    +0.000, E1   +45.850, E3 +414375.281}
SPL {X  -165.650, Y  +486.159, Z    +0.000, E1   +44.975, E3 +414388.826}
SPL {X  -165.650, Y  +482.261, Z    +0.000, E1   +43.960, E3 +414402.635}
SPL {X  -165.650, Y  +478.467, Z    +0.000, E1   +43.371, E3 +414414.463}
SPL {X  -165.650, Y  +474.990, Z    +0.000, E1   +42.535, E3 +414426.814}
SPL {X  -165.650, Y  +471.308, Z    +0.000, E1   +41.710, E3 +414440.320}
SPL {X  -165.650, Y  +467.130, Z    +0.000, E1   +40.624, E3 +414456.445}
SPL {X  -165.650, Y  +463.869, Z    +0.000, E1   +39.839, E3 +414468.913}
SPL {X  -165.650, Y  +462.171, Z    +0.000, E1   +38.860, E3 +414479.092}
SPL {X  -165.650, Y  +457.119, Z    +0.000, E1   +39.087, E3 +414490.470}
SPL {X  -165.650, Y  +452.884, Z    +0.000, E1   +39.185, E3 +414500.518}
SPL {X  -165.650, Y  +449.593, Z    +0.000, E1   +38.852, E3 +414510.813}
SPL {X  -165.650, Y  +445.147, Z    +0.000, E1   +39.088, E3 +414520.635}
SPL {X  -165.650, Y  +439.751, Z    +0.000, E1   +39.254, E3 +414533.252}
SPL {X  -165.650, Y  +435.510, Z    +0.000, E1   +39.051, E3 +414545.064}
SPL {X  -165.650, Y  +430.832, Z    +0.000, E1   +39.105, E3 +414556.520}
SPL {X  -165.650, Y  +426.072, Z    +0.000, E1   +39.194, E3 +414567.943}
SPL {X  -165.650, Y  +422.372, Z    +0.000, E1   +38.952, E3 +414578.679}
SPL {X  -165.650, Y  +417.591, Z    +0.000, E1   +39.157, E3 +414589.532}
SPL {X  -165.650, Y  +412.842, Z    +0.000, E1   +39.072, E3 +414602.031}
SPL {X  -165.650, Y  +407.612, Z    +0.000, E1   +39.068, E3 +414615.204}
SPL {X  -165.650, Y  +402.767, Z    +0.000, E1   +39.122, E3 +414627.059}
SPL {X  -165.650, Y  +398.352, Z    +0.000, E1   +39.113, E3 +414638.212}
SPL {X  -165.650, Y  +393.915, Z    +0.000, E1   +39.126, E3 +414649.289}
SPL {X  -165.650, Y  +389.523, Z    +0.000, E1   +39.115, E3 +414660.399}
SPL {X  -165.650, Y  +384.404, Z    +0.000, E1   +39.147, E3 +414673.135}
SPL {X  -165.650, Y  +380.058, Z    +0.000, E1   +39.073, E3 +414684.422}
SPL {X  -165.624, Y  +375.547, Z    +0.000, E1   +39.047, E3 +414696.021}
SPL {X  -165.438, Y  +370.129, Z    +0.000, E1   +39.090, E3 +414709.407}
SPL {X  -165.143, Y  +365.555, Z    +0.000, E1   +39.161, E3 +414720.379}
SPL {X  -164.909, Y  +362.853, Z    +0.000, E1   +38.709, E3 +414729.926}
SPL {X  -164.359, Y  +357.858, Z    +0.000, E1   +39.066, E3 +414740.389}
SPL {X  -163.818, Y  +353.935, Z    +0.000, E1   +38.811, E3 +414751.783}
SPL {X  -163.055, Y  +349.296, Z    +0.000, E1   +38.669, E3 +414764.288}
SPL {X  -162.319, Y  +345.445, Z    +0.000, E1   +38.490, E3 +414774.983}
SPL {X  -161.279, Y  +340.696, Z    +0.000, E1   +38.442, E3 +414787.311}
SPL {X  -160.251, Y  +336.552, Z    +0.000, E1   +38.166, E3 +414799.177}
SPL {X  -151.400, Y  +311.284, Z    +0.000, E1   +46.597, E3 +414806.900}
SPL {X  -146.894, Y  +301.936, Z    +0.000, E1   +40.559, E3 +414880.064}
ENDSPLINE

SPLINE
SPL {X  -154.092, Y  +317.709, Z    +0.000, E1   +32.342, E3 +414949.189}
SPL {X  -161.950, Y  +343.684, Z    +0.000, E1   +21.785, E3 +414926.028}
SPL {X  -164.623, Y  +360.087, Z    +0.000, E1   +13.426, E3 +414934.679}
SPL {X  -165.588, Y  +373.983, Z    +0.000, E1    +5.738, E3 +414927.455}
SPL {X  -165.650, Y  +380.761, Z    +0.000, E1    +1.351, E3 +414929.180}
SPL {X  -165.650, Y  +386.484, Z    +0.000, E1    -2.972, E3 +414927.187}
SPL {X  -165.650, Y  +391.786, Z    +0.000, E1    -7.566, E3 +414929.582}
SPL {X  -165.650, Y  +399.284, Z    +0.000, E1   -15.403, E3 +414924.767}
SPL {X  -165.650, Y  +409.824, Z    +0.000, E1   -26.455, E3 +414922.646}
SPL {X  -165.650, Y  +437.337, Z    +0.000, E1   -46.817, E3 +414925.281}
SPL {X  -165.650, Y  +450.640, Z    +0.000, E1   -46.274, E3 +414947.303}
SPL {X  -165.650, Y  +484.108, Z    +0.000, E1   -48.531, E3 +414992.082}
ENDSPLINE

SPLINE
SPL {X  -165.650, Y  +465.194, Z    +0.000, E1   -39.630, E3 +415003.950}
ENDSPLINE

SPLINE
SPL {X  -165.650, Y  +465.900, Z    +0.000, E1   -37.888, E3 +415016.653}
SPL {X  -165.650, Y  +471.256, Z    +0.000, E1   -37.789, E3 +415031.220}
SPL {X  -165.650, Y  +477.269, Z    +0.000, E1   -37.921, E3 +415046.437}
SPL {X  -165.650, Y  +483.881, Z    +0.000, E1   -37.934, E3 +415063.629}
SPL {X  -165.650, Y  +489.657, Z    +0.000, E1   -37.855, E3 +415079.290}
SPL {X  -165.650, Y  +496.067, Z    +0.000, E1   -37.879, E3 +415096.079}
SPL {X  -165.650, Y  +502.007, Z    +0.000, E1   -37.899, E3 +415111.461}
SPL {X  -165.650, Y  +506.838, Z    +0.000, E1   -38.018, E3 +415123.358}
SPL {X  -165.650, Y  +510.962, Z    +0.000, E1   -37.876, E3 +415135.072}
SPL {X  -165.650, Y  +513.924, Z    +0.000, E1   -37.557, E3 +415144.739}
SPL {X  -165.650, Y  +519.541, Z    +0.000, E1   -37.994, E3 +415157.074}
SPL {X  -165.650, Y  +524.168, Z    +0.000, E1   -37.816, E3 +415170.129}
SPL {X  -165.650, Y  +528.532, Z    +0.000, E1   -37.895, E3 +415181.195}
SPL {X  -165.650, Y  +532.864, Z    +0.000, E1   -37.846, E3 +415192.837}
SPL {X  -165.650, Y  +537.279, Z    +0.000, E1   -37.980, E3 +415203.660}
SPL {X  -165.650, Y  +540.651, Z    +0.000, E1   -37.651, E3 +415214.462}
SPL {X  -165.650, Y  +545.726, Z    +0.000, E1   -37.963, E3 +415226.028}
SPL {X  -165.650, Y  +550.427, Z    +0.000, E1   -37.784, E3 +415239.445}
SPL {X  -165.650, Y  +556.372, Z    +0.000, E1   -37.998, E3 +415253.842}
SPL {X  -165.650, Y  +561.478, Z    +0.000, E1   -37.846, E3 +415268.089}
SPL {X  -165.650, Y  +566.625, Z    +0.000, E1   -37.932, E3 +415281.118}
SPL {X  -165.650, Y  +571.305, Z    +0.000, E1   -37.718, E3 +415294.756}
SPL {X  -165.650, Y  +577.754, Z    +0.000, E1   -38.006, E3 +415310.047}
SPL {X  -165.650, Y  +583.042, Z    +0.000, E1   -37.879, E3 +415324.590}
SPL {X  -165.650, Y  +587.643, Z    +0.000, E1   -37.879, E3 +415336.669}
SPL {X  -165.650, Y  +592.833, Z    +0.000, E1   -37.896, E3 +415350.317}
SPL {X  -165.650, Y  +597.119, Z    +0.000, E1   -37.642, E3 +415363.046}
SPL {X  -165.650, Y  +602.808, Z    +0.000, E1   -37.983, E3 +415376.052}
SPL {X  -165.650, Y  +607.937, Z    +0.000, E1   -37.862, E3 +415390.214}
SPL {X  -165.650, Y  +614.056, Z    +0.000, E1   -37.933, E3 +415405.984}
SPL {X  -165.650, Y  +619.142, Z    +0.000, E1   -37.954, E3 +415419.003}
SPL {X  -165.650, Y  +622.884, Z    +0.000, E1   -37.770, E3 +415430.046}
SPL {X  -165.650, Y  +627.016, Z    +0.000, E1   -37.897, E3 +415440.084}
SPL {X  -165.650, Y  +630.421, Z    +0.000, E1   -38.020, E3 +415448.247}
SPL {X  -165.650, Y  +633.686, Z    +0.000, E1   -37.760, E3 +415458.491}
SPL {X  -165.650, Y  +638.669, Z    +0.000, E1   -37.941, E3 +415470.498}
SPL {X  -165.650, Y  +643.208, Z    +0.000, E1   -37.786, E3 +415483.414}
SPL {X  -165.650, Y  +649.293, Z    +0.000, E1   -37.920, E3 +415498.704}
SPL {X  -165.650, Y  +654.711, Z    +0.000, E1   -37.888, E3 +415513.026}
SPL {X  -165.650, Y  +658.674, Z    +0.000, E1   -37.902, E3 +415523.294}
SPL {X  -165.650, Y  +661.754, Z    +0.000, E1   -37.878, E3 +415531.530}
SPL {X  -165.650, Y  +665.663, Z    +0.000, E1   -37.913, E3 +415541.631}
SPL {X  -165.650, Y  +669.913, Z    +0.000, E1   -37.905, E3 +415552.833}
SPL {X  -165.650, Y  +674.729, Z    +0.000, E1   -37.860, E3 +415565.843}
SPL {X  -165.591, Y  +679.928, Z    +0.000, E1   -37.818, E3 +415579.760}
SPL {X  -165.340, Y  +685.624, Z    +0.000, E1   -37.900, E3 +415594.295}
SPL {X  -165.010, Y  +690.051, Z    +0.000, E1   -37.675, E3 +415607.226}
SPL {X  -164.652, Y  +693.652, Z    +0.000, E1   -37.750, E3 +415616.156}
SPL {X  -164.143, Y  +697.797, Z    +0.000, E1   -37.636, E3 +415627.975}
SPL {X  -163.447, Y  +702.423, Z    +0.000, E1   -37.496, E3 +415640.784}
SPL {X  -162.809, Y  +706.049, Z    +0.000, E1   -37.384, E3 +415651.054}
SPL {X  -161.803, Y  +710.992, Z    +0.000, E1   -37.315, E3 +415664.519}
SPL {X  -160.993, Y  +714.501, Z    +0.000, E1   -36.839, E3 +415676.395}
SPL {X  -159.156, Y  +721.427, Z    +0.000, E1   -38.526, E3 +415684.473}
SPL {X  -144.831, Y  +755.898, Z    +0.000, E1   -42.981, E3 +415745.889}
ENDSPLINE

SPLINE
SPL {X  -153.047, Y  +738.876, Z    +0.000, E1   -33.363, E3 +415828.104}
SPL {X  -162.649, Y  +706.888, Z    +0.000, E1   -19.911, E3 +415817.466}
SPL {X  -165.011, Y  +690.033, Z    +0.000, E1   -11.292, E3 +415813.700}
SPL {X  -165.581, Y  +680.273, Z    +0.000, E1    -5.775, E3 +415809.499}
SPL {X  -165.650, Y  +674.660, Z    +0.000, E1    -2.196, E3 +415810.166}
SPL {X  -165.650, Y  +669.932, Z    +0.000, E1    +1.173, E3 +415808.742}
SPL {X  -165.650, Y  +665.412, Z    +0.000, E1    +4.953, E3 +415807.921}
SPL {X  -165.650, Y  +658.891, Z    +0.000, E1   +11.031, E3 +415808.232}
SPL {X  -165.650, Y  +649.186, Z    +0.000, E1   +20.530, E3 +415809.492}
SPL {X  -165.650, Y  +637.823, Z    +0.000, E1   +39.473, E3 +415789.088}
SPL {X  -165.650, Y  +613.283, Z    +0.000, E1   +49.826, E3 +415804.655}
SPL {X  -165.650, Y  +609.693, Z    +0.000, E1   +42.113, E3 +415832.789}
SPL {X  -165.650, Y  +571.120, Z    +0.000, E1   +47.704, E3 +415877.599}
ENDSPLINE

SPLINE
SPL {X  -165.650, Y  +586.477, Z    +0.000, E1   +39.172, E3 +415894.143}
ENDSPLINE

SPLINE
SPL {X  -165.650, Y  +581.917, Z    +0.000, E1   +39.019, E3 +415906.545}
SPL {X  -165.650, Y  +577.218, Z    +0.000, E1   +38.911, E3 +415919.085}
SPL {X  -165.650, Y  +571.720, Z    +0.000, E1   +39.004, E3 +415932.477}
SPL {X  -165.650, Y  +565.656, Z    +0.000, E1   +39.042, E3 +415947.586}
SPL {X  -165.650, Y  +560.333, Z    +0.000, E1   +38.995, E3 +415961.215}
SPL {X  -165.650, Y  +554.558, Z    +0.000, E1   +39.065, E3 +415975.503}
SPL {X  -165.650, Y  +548.147, Z    +0.000, E1   +39.104, E3 +415991.360}
SPL {X  -165.650, Y  +526.098, Z    +0.000, E1   +45.792, E3 +416001.179}
SPL {X  -165.650, Y  +510.223, Z    +0.000, E1   +49.521, E3 +416008.576}
SPL {X  -165.650, Y  +506.429, Z    +0.000, E1   +48.913, E3 +416018.989}
SPL {X  -165.650, Y  +501.394, Z    +0.000, E1   +48.110, E3 +416032.968}
SPL {X  -165.650, Y  +497.138, Z    +0.000, E1   +47.280, E3 +416045.664}
SPL {X  -165.650, Y  +493.273, Z    +0.000, E1   +46.518, E3 +416057.645}
SPL {X  -165.650, Y  +489.140, Z    +0.000, E1   +45.675, E3 +416070.772}
SPL {X  -165.650, Y  +485.420, Z    +0.000, E1   +44.711, E3 +416083.991}
SPL {X  -165.650, Y  +482.261, Z    +0.000, E1   +43.960, E3 +416094.943}
SPL {X  -165.650, Y  +479.614, Z    +0.000, E1   +43.544, E3 +416103.077}
SPL {X  -165.650, Y  +475.837, Z    +0.000, E1   +42.787, E3 +416115.930}
SPL {X  -165.650, Y  +472.413, Z    +0.000, E1   +41.852, E3 +416129.044}
SPL {X  -165.650, Y  +468.649, Z    +0.000, E1   +41.090, E3 +416142.408}
SPL {X  -165.650, Y  +464.675, Z    +0.000, E1   +40.045, E3 +416158.186}
SPL {X  -165.650, Y  +462.171, Z    +0.000, E1   +38.860, E3 +416171.400}
SPL {X  -165.650, Y  +457.119, Z    +0.000, E1   +39.087, E3 +416182.778}
SPL {X  -165.650, Y  +452.884, Z    +0.000, E1   +39.185, E3 +416192.826}
SPL {X  -165.650, Y  +449.593, Z    +0.000, E1   +38.852, E3 +416203.121}
SPL {X  -165.650, Y  +445.147, Z    +0.000, E1   +39.088, E3 +416212.943}
SPL {X  -165.650, Y  +439.751, Z    +0.000, E1   +39.254, E3 +416225.560}
SPL {X  -165.650, Y  +435.510, Z    +0.000, E1   +39.051, E3 +416237.371}
SPL {X  -165.650, Y  +430.832, Z    +0.000, E1   +39.105, E3 +416248.828}
SPL {X  -165.650, Y  +426.072, Z    +0.000, E1   +39.194, E3 +416260.251}
SPL {X  -165.650, Y  +422.372, Z    +0.000, E1   +38.952, E3 +416270.987}
SPL {X  -165.650, Y  +417.591, Z    +0.000, E1   +39.157, E3 +416281.840}
SPL {X  -165.650, Y  +412.842, Z    +0.000, E1   +39.072, E3 +416294.339}
SPL {X  -165.650, Y  +407.612, Z    +0.000, E1   +39.068, E3 +416307.511}
SPL {X  -165.650, Y  +402.767, Z    +0.000, E1   +39.122, E3 +416319.367}
SPL {X  -165.650, Y  +398.352, Z    +0.000, E1   +39.113, E3 +416330.520}
SPL {X  -165.650, Y  +393.915, Z    +0.000, E1   +39.126, E3 +416341.597}
SPL {X  -165.650, Y  +388.386, Z    +0.000, E1   +39.140, E3 +416355.547}
SPL {X  -165.650, Y  +383.342, Z    +0.000, E1   +39.144, E3 +416368.033}
SPL {X  -165.650, Y  +378.675, Z    +0.000, E1   +39.090, E3 +416380.251}
SPL {X  -165.597, Y  +374.311, Z    +0.000, E1   +39.013, E3 +416391.537}
SPL {X  -165.438, Y  +370.129, Z    +0.000, E1   +39.090, E3 +416401.715}
SPL {X  -165.143, Y  +365.555, Z    +0.000, E1   +39.161, E3 +416412.687}
SPL {X  -164.909, Y  +362.853, Z    +0.000, E1   +38.709, E3 +416422.233}
SPL {X  -164.359, Y  +357.858, Z    +0.000, E1   +39.066, E3 +416432.696}
SPL {X  -163.818, Y  +353.935, Z    +0.000, E1   +38.811, E3 +416444.090}
SPL {X  -163.055, Y  +349.296, Z    +0.000, E1   +38.669, E3 +416456.596}
SPL {X  -162.319, Y  +345.445, Z    +0.000, E1   +38.490, E3 +416467.291}
SPL {X  -161.279, Y  +340.696, Z    +0.000, E1   +38.442, E3 +416479.619}
SPL {X  -160.251, Y  +336.552, Z    +0.000, E1   +38.166, E3 +416491.484}
SPL {X  -151.400, Y  +311.284, Z    +0.000, E1   +46.597, E3 +416499.208}
SPL {X  -146.894, Y  +301.936, Z    +0.000, E1   +40.559, E3 +416572.372}
ENDSPLINE

SPLINE
SPL {X  -154.092, Y  +317.709, Z    +0.000, E1   +32.342, E3 +416641.497}
SPL {X  -161.950, Y  +343.684, Z    +0.000, E1   +21.785, E3 +416618.336}
SPL {X  -164.623, Y  +360.087, Z    +0.000, E1   +13.426, E3 +416626.986}
SPL {X  -165.489, Y  +371.187, Z    +0.000, E1    +7.370, E3 +416617.827}
SPL {X  -165.621, Y  +375.403, Z    +0.000, E1    +4.810, E3 +416620.725}
SPL {X  -165.650, Y  +380.761, Z    +0.000, E1    +1.351, E3 +416621.487}
SPL {X  -165.650, Y  +386.484, Z    +0.000, E1    -2.972, E3 +416619.494}
SPL {X  -165.650, Y  +392.905, Z    +0.000, E1    -8.557, E3 +416621.548}
SPL {X  -165.650, Y  +404.146, Z    +0.000, E1   -20.514, E3 +416616.278}
SPL {X  -165.650, Y  +412.709, Z    +0.000, E1   -30.621, E3 +416611.242}
SPL {X  -165.650, Y  +437.337, Z    +0.000, E1   -46.817, E3 +416617.589}
SPL {X  -165.650, Y  +450.640, Z    +0.000, E1   -46.274, E3 +416639.611}
SPL {X  -165.650, Y  +484.108, Z    +0.000, E1   -48.531, E3 +416684.390}
ENDSPLINE

SPLINE
SPL {X  -165.650, Y  +464.452, Z    +0.000, E1   -38.833, E3 +416699.451}
ENDSPLINE

SPLINE
SPL {X  -165.650, Y  +467.011, Z    +0.000, E1   -37.866, E3 +416711.874}
SPL {X  -165.650, Y  +471.256, Z    +0.000, E1   -37.789, E3 +416723.528}
SPL {X  -165.650, Y  +475.981, Z    +0.000, E1   -37.909, E3 +416735.251}
SPL {X  -165.650, Y  +481.142, Z    +0.000, E1   -37.875, E3 +416749.071}
SPL {X  -165.650, Y  +487.016, Z    +0.000, E1   -37.964, E3 +416763.977}
SPL {X  -165.650, Y  +492.473, Z    +0.000, E1   -37.882, E3 +416778.773}
SPL {X  -165.650, Y  +496.967, Z    +0.000, E1   -37.731, E3 +416791.480}
SPL {X  -165.650, Y  +502.007, Z    +0.000, E1   -37.899, E3 +416803.769}
SPL {X  -165.650, Y  +507.602, Z    +0.000, E1   -37.863, E3 +416818.799}
SPL {X  -165.650, Y  +513.428, Z    +0.000, E1   -37.892, E3 +416833.865}
SPL {X  -165.650, Y  +518.534, Z    +0.000, E1   -37.976, E3 +416846.728}
SPL {X  -165.650, Y  +523.331, Z    +0.000, E1   -37.880, E3 +416859.950}
SPL {X  -165.650, Y  +528.532, Z    +0.000, E1   -37.895, E3 +416873.503}
SPL {X  -165.650, Y  +532.864, Z    +0.000, E1   -37.846, E3 +416885.145}
SPL {X  -165.650, Y  +537.279, Z    +0.000, E1   -37.980, E3 +416895.967}
SPL {X  -165.650, Y  +540.651, Z    +0.000, E1   -37.651, E3 +416906.770}
SPL {X  -165.650, Y  +545.726, Z    +0.000, E1   -37.963, E3 +416918.335}
SPL {X  -165.650, Y  +550.427, Z    +0.000, E1   -37.784, E3 +416931.753}
SPL {X  -165.650, Y  +554.659, Z    +0.000, E1   -37.927, E3 +416941.937}
SPL {X  -165.650, Y  +557.856, Z    +0.000, E1   -37.998, E3 +416949.887}
SPL {X  -165.650, Y  +562.748, Z    +0.000, E1   -37.890, E3 +416963.630}
SPL {X  -165.650, Y  +567.848, Z    +0.000, E1   -37.954, E3 +416976.402}
SPL {X  -165.650, Y  +571.305, Z    +0.000, E1   -37.718, E3 +416987.063}
SPL {X  -165.650, Y  +577.754, Z    +0.000, E1   -38.006, E3 +417002.355}
SPL {X  -165.650, Y  +583.042, Z    +0.000, E1   -37.879, E3 +417016.898}
SPL {X  -165.650, Y  +587.643, Z    +0.000, E1   -37.879, E3 +417028.976}
SPL {X  -165.650, Y  +592.833, Z    +0.000, E1   -37.896, E3 +417042.625}
SPL {X  -165.650, Y  +599.187, Z    +0.000, E1   -37.841, E3 +417059.763}
SPL {X  -165.650, Y  +604.276, Z    +0.000, E1   -37.917, E3 +417072.451}
SPL {X  -165.650, Y  +607.937, Z    +0.000, E1   -37.862, E3 +417082.521}
SPL {X  -165.650, Y  +612.863, Z    +0.000, E1   -37.857, E3 +417095.494}
SPL {X  -165.650, Y  +618.208, Z    +0.000, E1   -37.992, E3 +417108.736}
SPL {X  -165.650, Y  +622.884, Z    +0.000, E1   -37.770, E3 +417122.353}
SPL {X  -165.650, Y  +628.759, Z    +0.000, E1   -37.993, E3 +417136.523}
SPL {X  -165.650, Y  +633.686, Z    +0.000, E1   -37.760, E3 +417150.799}
SPL {X  -165.650, Y  +638.669, Z    +0.000, E1   -37.941, E3 +417162.805}
SPL {X  -165.650, Y  +644.441, Z    +0.000, E1   -37.838, E3 +417178.820}
SPL {X  -165.650, Y  +650.450, Z    +0.000, E1   -37.924, E3 +417193.899}
SPL {X  -165.650, Y  +654.711, Z    +0.000, E1   -37.888, E3 +417205.333}
SPL {X  -165.650, Y  +660.285, Z    +0.000, E1   -37.928, E3 +417219.852}
SPL {X  -165.650, Y  +665.663, Z    +0.000, E1   -37.913, E3 +417233.939}
SPL {X  -165.650, Y  +671.321, Z    +0.000, E1   -37.904, E3 +417249.040}
SPL {X  -165.649, Y  +676.172, Z    +0.000, E1   -37.873, E3 +417261.737}
SPL {X  -165.554, Y  +681.132, Z    +0.000, E1   -37.883, E3 +417274.985}
SPL {X  -165.277, Y  +686.615, Z    +0.000, E1   -37.853, E3 +417289.367}
SPL {X  -165.010, Y  +690.051, Z    +0.000, E1   -37.675, E3 +417299.533}
SPL {X  -164.652, Y  +693.652, Z    +0.000, E1   -37.750, E3 +417308.464}
SPL {X  -164.143, Y  +697.797, Z    +0.000, E1   -37.636, E3 +417320.283}
SPL {X  -163.447, Y  +702.423, Z    +0.000, E1   -37.496, E3 +417333.091}
SPL {X  -162.809, Y  +706.049, Z    +0.000, E1   -37.384, E3 +417343.362}
SPL {X  -162.124, Y  +709.497, Z    +0.000, E1   -37.325, E3 +417352.684}
SPL {X  -161.242, Y  +713.462, Z    +0.000, E1   -37.074, E3 +417364.805}
SPL {X  -159.156, Y  +721.427, Z    +0.000, E1   -38.526, E3 +417376.781}
SPL {X  -144.831, Y  +755.898, Z    +0.000, E1   -42.981, E3 +417438.197}
ENDSPLINE

SPLINE
SPL {X  -153.047, Y  +738.876, Z    +0.000, E1   -33.363, E3 +417520.412}
SPL {X  -162.649, Y  +706.888, Z    +0.000, E1   -19.911, E3 +417509.774}
SPL {X  -165.011, Y  +690.033, Z    +0.000, E1   -11.292, E3 +417506.008}
SPL {X  -165.581, Y  +680.273, Z    +0.000, E1    -5.775, E3 +417501.806}
SPL {X  -165.650, Y  +673.781, Z    +0.000, E1    -1.642, E3 +417501.049}
SPL {X  -165.650, Y  +669.471, Z    +0.000, E1    +1.546, E3 +417502.204}
SPL {X  -165.650, Y  +665.412, Z    +0.000, E1    +4.953, E3 +417500.229}
SPL {X  -165.650, Y  +660.335, Z    +0.000, E1    +9.682, E3 +417500.747}
SPL {X  -165.650, Y  +650.970, Z    +0.000, E1   +18.783, E3 +417501.294}
SPL {X  -165.650, Y  +637.823, Z    +0.000, E1   +39.473, E3 +417481.396}
SPL {X  -165.650, Y  +614.460, Z    +0.000, E1   +51.116, E3 +417492.264}
SPL {X  -165.650, Y  +609.746, Z    +0.000, E1   +42.762, E3 +417522.922}
SPL {X  -165.650, Y  +571.120, Z    +0.000, E1   +47.704, E3 +417569.906}
ENDSPLINE

SPLINE
SPL {X  -165.650, Y  +586.477, Z    +0.000, E1   +39.172, E3 +417586.451}
ENDSPLINE

SPLINE
SPL {X  -165.650, Y  +581.917, Z    +0.000, E1   +39.019, E3 +417598.853}
SPL {X  -165.650, Y  +577.218, Z    +0.000, E1   +38.911, E3 +417611.393}
SPL {X  -165.650, Y  +571.720, Z    +0.000, E1   +39.004, E3 +417624.785}
SPL {X  -165.650, Y  +565.656, Z    +0.000, E1   +39.042, E3 +417639.894}
SPL {X  -165.650, Y  +560.333, Z    +0.000, E1   +38.995, E3 +417653.522}
SPL {X  -165.650, Y  +554.558, Z    +0.000, E1   +39.065, E3 +417667.811}
SPL {X  -165.650, Y  +548.147, Z    +0.000, E1   +39.104, E3 +417683.667}
SPL {X  -165.650, Y  +526.098, Z    +0.000, E1   +45.792, E3 +417693.486}
SPL {X  -165.650, Y  +510.223, Z    +0.000, E1   +49.521, E3 +417700.883}
SPL {X  -165.650, Y  +506.429, Z    +0.000, E1   +48.913, E3 +417711.296}
SPL {X  -165.650, Y  +501.394, Z    +0.000, E1   +48.110, E3 +417725.275}
SPL {X  -165.650, Y  +497.138, Z    +0.000, E1   +47.280, E3 +417737.971}
SPL {X  -165.650, Y  +493.273, Z    +0.000, E1   +46.518, E3 +417749.952}
SPL {X  -165.650, Y  +489.140, Z    +0.000, E1   +45.675, E3 +417763.080}
SPL {X  -165.650, Y  +485.420, Z    +0.000, E1   +44.711, E3 +417776.299}
SPL {X  -165.650, Y  +480.756, Z    +0.000, E1   +43.779, E3 +417791.777}
SPL {X  -165.650, Y  +475.837, Z    +0.000, E1   +42.787, E3 +417808.237}
SPL {X  -165.650, Y  +472.413, Z    +0.000, E1   +41.852, E3 +417821.352}
SPL {X  -165.650, Y  +468.649, Z    +0.000, E1   +41.090, E3 +417834.716}
SPL {X  -165.650, Y  +464.675, Z    +0.000, E1   +40.045, E3 +417850.493}
SPL {X  -165.650, Y  +462.171, Z    +0.000, E1   +38.860, E3 +417863.708}
SPL {X  -165.650, Y  +457.119, Z    +0.000, E1   +39.087, E3 +417875.086}
SPL {X  -165.650, Y  +452.884, Z    +0.000, E1   +39.185, E3 +417885.134}
SPL {X  -165.650, Y  +449.593, Z    +0.000, E1   +38.852, E3 +417895.428}
SPL {X  -165.650, Y  +445.147, Z    +0.000, E1   +39.088, E3 +417905.251}
SPL {X  -165.650, Y  +439.751, Z    +0.000, E1   +39.254, E3 +417917.868}
SPL {X  -165.650, Y  +435.510, Z    +0.000, E1   +39.051, E3 +417929.679}
SPL {X  -165.650, Y  +430.832, Z    +0.000, E1   +39.105, E3 +417941.136}
SPL {X  -165.650, Y  +426.072, Z    +0.000, E1   +39.194, E3 +417952.559}
SPL {X  -165.650, Y  +422.372, Z    +0.000, E1   +38.952, E3 +417963.295}
SPL {X  -165.650, Y  +416.355, Z    +0.000, E1   +39.151, E3 +417977.454}
SPL {X  -165.650, Y  +408.927, Z    +0.000, E1   +39.115, E3 +417996.413}
SPL {X  -165.650, Y  +402.767, Z    +0.000, E1   +39.122, E3 +418011.674}
SPL {X  -165.650, Y  +398.352, Z    +0.000, E1   +39.113, E3 +418022.827}
SPL {X  -165.650, Y  +393.915, Z    +0.000, E1   +39.126, E3 +418033.904}
SPL {X  -165.650, Y  +389.523, Z    +0.000, E1   +39.115, E3 +418045.015}
SPL {X  -165.650, Y  +384.404, Z    +0.000, E1   +39.147, E3 +418057.750}
SPL {X  -165.650, Y  +378.675, Z    +0.000, E1   +39.090, E3 +418072.559}
SPL {X  -165.597, Y  +374.311, Z    +0.000, E1   +39.013, E3 +418083.844}
SPL {X  -165.438, Y  +370.129, Z    +0.000, E1   +39.090, E3 +418094.022}
SPL {X  -165.143, Y  +365.555, Z    +0.000, E1   +39.161, E3 +418104.995}
SPL {X  -164.909, Y  +362.853, Z    +0.000, E1   +38.709, E3 +418114.541}
SPL {X  -164.359, Y  +357.858, Z    +0.000, E1   +39.066, E3 +418125.004}
SPL {X  -163.818, Y  +353.935, Z    +0.000, E1   +38.811, E3 +418136.398}
SPL {X  -163.055, Y  +349.296, Z    +0.000, E1   +38.669, E3 +418148.903}
SPL {X  -162.319, Y  +345.445, Z    +0.000, E1   +38.490, E3 +418159.599}
SPL {X  -161.279, Y  +340.696, Z    +0.000, E1   +38.442, E3 +418171.926}
SPL {X  -160.251, Y  +336.552, Z    +0.000, E1   +38.166, E3 +418183.792}
SPL {X  -151.400, Y  +311.284, Z    +0.000, E1   +46.597, E3 +418191.515}
SPL {X  -146.894, Y  +301.936, Z    +0.000, E1   +40.559, E3 +418264.680}
ENDSPLINE

SPLINE
SPL {X  -154.092, Y  +317.709, Z    +0.000, E1   +32.342, E3 +418333.804}
SPL {X  -161.950, Y  +343.684, Z    +0.000, E1   +21.785, E3 +418310.644}
SPL {X  -164.623, Y  +360.087, Z    +0.000, E1   +13.426, E3 +418319.294}
SPL {X  -165.588, Y  +373.983, Z    +0.000, E1    +5.738, E3 +418312.071}
SPL {X  -165.650, Y  +380.761, Z    +0.000, E1    +1.351, E3 +418313.795}
SPL {X  -165.650, Y  +385.186, Z    +0.000, E1    -1.985, E3 +418312.280}
SPL {X  -165.650, Y  +387.866, Z    +0.000, E1    -4.228, E3 +418311.293}
SPL {X  -165.650, Y  +391.786, Z    +0.000, E1    -7.566, E3 +418314.197}
SPL {X  -165.650, Y  +395.964, Z    +0.000, E1   -11.741, E3 +418312.921}
SPL {X  -165.650, Y  +404.146, Z    +0.000, E1   -20.514, E3 +418308.586}
SPL {X  -165.650, Y  +416.920, Z    +0.000, E1   -34.832, E3 +418302.549}
SPL {X  -165.650, Y  +445.455, Z    +0.000, E1   -46.044, E3 +418324.640}
SPL {X  -165.650, Y  +459.839, Z    +0.000, E1   -48.128, E3 +418339.706}
SPL {X  -165.650, Y  +484.108, Z    +0.000, E1   -48.531, E3 +418376.698}
ENDSPLINE

SPLINE
SPL {X  -165.650, Y  +465.194, Z    +0.000, E1   -39.630, E3 +418388.566}
ENDSPLINE

